IF R_HMICommand.Q THEN
    IF MainPMLControl_Simplified.ResetPressed AND
       MainPMLControl_Simplified.ResetPermissive AND
       MainPMLControl_Standard.CurrentState = E_PMLState.ePMLState_Aborted THEN
        ipModule.ChangeState(Tc3_PackML_V2.E_PMLCommand.ePMLCommand_Clear);
    ELSIF MainPMLControl_Simplified.ResetPressed AND MainPMLControl_Simplified.ResetPermissive THEN
        ipModule.ChangeState(Tc3_PackML_V2.E_PMLCommand.ePMLCommand_Reset);
    ELSIF MainPMLControl_Simplified.StartPressed AND MainPMLControl_Simplified.StartPermissive THEN
        IF MainPMLControl_Standard.CurrentState = Tc3_PackML_V2.E_PMLState.ePMLState_Idle THEN
            ipModule.ChangeState(Tc3_PackML_V2.E_PMLCommand.ePMLCommand_Start);
        ELSIF MainPMLControl_Standard.CurrentState = Tc3_PackML_V2.E_PMLState.ePMLState_Held THEN
            ipModule.ChangeState(Tc3_PackML_V2.E_PMLCommand.ePMLCommand_Unhold);
        ELSIF MainPMLControl_Standard.CurrentState = Tc3_PackML_V2.E_PMLState.ePMLState_Suspended THEN
            ipModule.ChangeState(Tc3_PackML_V2.E_PMLCommand.ePMLCommand_Unsuspend);
        END_IF
    ELSIF MainPMLControl_Simplified.StopPressed AND MainPMLControl_Simplified.StopPermissive THEN
        ipModule.ChangeState(Tc3_PackML_V2.E_PMLCommand.ePMLCommand_Stop);
    ELSIF MainPMLControl_Simplified.AbortPressed AND MainPMLControl_Simplified.AbortPermissive THEN
        ipModule.ChangeState(Tc3_PackML_V2.E_PMLCommand.ePMLCommand_Abort);
    ELSIF MainPMLControl_Simplified.HoldPressed AND MainPMLControl_Simplified.HoldPermissive THEN
        ipModule.ChangeState(Tc3_PackML_V2.E_PMLCommand.ePMLCommand_Hold);
    ELSIF ipModule.StateCommand <> MainPMLControl_Standard.StateCommand THEN
        ipModule.StateCommand := MainPMLControl_Standard.StateCommand;
    ELSIF ipModule.ModeCommand <> MainPMLControl_Standard.ModeCommand THEN
        ipModule.ModeCommand := MainPMLControl_Standard.ModeCommand;
    END_IF
END_IF

MainPMLControl_Simplified.StartPermissive := MainPMLControl_Standard.CurrentState = Tc3_PackML_V2.E_PMLState.ePMLState_Idle OR
                                             MainPMLControl_Standard.CurrentState = Tc3_PackML_V2.E_PMLState.ePMLState_Held OR
                                             MainPMLControl_Standard.CurrentState = Tc3_PackML_V2.E_PMLState.ePMLState_Suspended;

MainPMLControl_Simplified.HoldPermissive := MainPMLControl_Standard.CurrentState = Tc3_PackML_V2.E_PMLState.ePMLState_Execute OR
                                            MainPMLControl_Standard.CurrentState = Tc3_PackML_V2.E_PMLState.ePMLState_Unsuspending OR
                                            MainPMLControl_Standard.CurrentState = Tc3_PackML_V2.E_PMLState.ePMLState_Unholding;

MainPMLControl_Simplified.StopPermissive := MainPMLControl_Simplified.AbortPermissive :=
    MainPMLControl_Standard.CurrentState = Tc3_PackML_V2.E_PMLState.ePMLState_Held OR
    MainPMLControl_Standard.CurrentState = Tc3_PackML_V2.E_PMLState.ePMLState_Suspended OR
    MainPMLControl_Standard.CurrentState = Tc3_PackML_V2.E_PMLState.ePMLState_Idle;

MainPMLControl_Simplified.ResetPermissive := MainPMLControl_Standard.CurrentState = Tc3_PackML_V2.E_PMLState.ePMLState_Complete OR
                                             MainPMLControl_Standard.CurrentState = Tc3_PackML_V2.E_PMLState.ePMLState_Stopped OR
                                             MainPMLControl_Standard.CurrentState = Tc3_PackML_V2.E_PMLState.ePMLState_Aborted;
END_METHOD

PROPERTY Control : SPT_BaseTypes.I_PackML_Control
SET
ipModule := Control;
END_SET
END_PROPERTY

METHOD FINAL ModeChanged
VAR_INPUT
    NewMode : SPT_BaseTypes.E_PMLUnitMode;
END_VAR
MainPMLControl_Standard.ModeCommand := NewMode;
END_METHOD

METHOD FINAL StateChanged
VAR_INPUT
    NewState : SPT_BaseTypes.E_PMLCommand;
END_VAR
MainPMLControl_Standard.StateCommand := NewState;
END_METHOD

PROPERTY ForceHoldRequested : Bool
GET
ForceHoldRequested := (MainPMLControl_Standard.CurrentState = Tc3_PackML_V2.E_PMLState.ePMLState_Unsuspending OR
                      MainPMLControl_Standard.CurrentState = Tc3_PackML_V2.E_PMLState.ePMLState_Unholding) AND
                      MainPMLControl_Simplified.HoldPressed;
END_GET
END_PROPERTY

METHOD FINAL Initialize : BOOL
IF Registered THEN
    Initialize := TRUE;
END_IF
END_METHOD

PROPERTY Registered : BOOL
GET
Registered := ipModule <> 0;
END_GET
END_PROPERTY

END_FUNCTION_BLOCK

// Machine/EquipmentModules/Functional Layer/FB_Carriage
FUNCTION_BLOCK FB_Carriage EXTENDS FB_EquipmentModule_SR
VAR
    // Sub module definitions here

    // List of sub modules

    ipSubModules_Init : ARRAY[1..Parameters_PackML_Base.MAX_NO_OF_SUBMODULES] OF I_PackML_BaseModule := [];

    // Component definitions here

    // Transporter components based on class diagram

    Pos                 : FB_Component_BasicSlaveAxis_SoE := (Name := 'Position');
    Pick                : FB_Component_BasicSlaveAxis_SoE := (Name := 'Pick');
    BoardPresentSensor1 : FB_DigitalSensor                := (Name := 'BoardPresentSensor1');
    BoardPresentSensor2 : FB_DigitalSensor                := (Name := 'BoardPresentSensor2');
    HomingSensor        : FB_DigitalSensor                := (Name := 'HomingSensor');

    //Alarms for this module

    Pick_TorqueControl          : SPT_Motion_Control.MC_TorqueControl;
    Pick_HomingInfo             : ST_HomingParams;
    Pick_TorqueReference AT %Q* : UINT  := 100;
    Pick_First_Torque           : LREAL := -30;
    Pick_Second_Torque          : LREAL := -20;
    Pick_Home_Torque            : LREAL := 35;
    Pick_Lag                    : LREAL := 8;
    Pick_Vel                    : LREAL := 1200;

    MoveStates    : ST_MoveStates;
    SpeedSelected : E_SpeedOptions := E_SpeedOptions.TESTING1;

    Execute_TorqueMove      : BOOL;
    _SensorOverride         : BOOL;
    _SensorIgnore           : BOOL;
    BoardsIgnoredCount      : USINT;
    BoardSecured_AfterStop  : BOOL;
    GrabTorqueNotCompleting : BOOL;
    ReleaseNotFinished      : BOOL;
    MoveIdleNotFinished     : BOOL;
END_VAR

VAR CONSTANT
    //reports 

    FAULT : INT := 1;

    //Alarms

    UNWIND_ALARM_COUNT    : INT   := 5;
    CARRIAGE_ALARMS_COUNT : USINT := 10;
END_VAR

VAR
	PickMotorCmds_Extra : ST_MotorControls_NonStandard;
	PosMotorCmds_Extra : ST_MotorControls_NonStandard;

    _TargetPos       : LREAL;
    _IdlePos         : REAL;
    _HoldingBoard    : BOOL;
    _TestPick        : BOOL;
    _BoardSecured    : BOOL;
    _BoardDataToPass : ST_BoardData;

    _CarriageCollisionCheckOK    : BOOL;
    _BoardCollisionCheckOK       : BOOL;
    _MoveClearActive             : BOOL;
    _BoardHeight                 : LREAL;
    _MoveState                   : E_MoveCarriageState;
    _MoveSubState                : UDINT;
    CarriageMovementRequestState : UDINT;

    _ClearOfCarriages      : BOOL;
    _ClearOfBoards         : BOOL;
    _ActuatorsOpen         : BOOL;
    _ActuatorsClosed       : BOOL;
    _MovementRequested     : BOOL;
    _OpenActuatorsRequest  : BOOL;
    _CloseActuatorsRequest : BOOL;

    MoveIdleState : USINT;

    HomeHardStop : BOOL;

    //Homing Options

    TorqueOptions : SPT_Motion_Control.ST_TorqueControlOptions;

    _PressPermissions : ST_MediatorInterface;

    _MasterAxisRef : REFERENCE TO SPT_Motion_Control.AXIS_REF;
    _AxisRef       : REFERENCE TO SPT_Motion_Control.AXIS_REF;

    Grab_State    : E_GrabState;
    Release_State : E_ReleaseState;

    LastBoardHeightGrabbed : LREAL := 100;
    ;

    CarriageAlarms : ARRAY[1..CARRIAGE_ALARMS_COUNT] OF FB_TcAlarm;
	
END_VAR

METHOD CyclicLogic
VAR_INPUT
END_VAR
IF NOT _InitComplete THEN
    _InitComplete := Initialize();
    RETURN;
END_IF

SUPER^.CyclicLogic();

//HMI control for EM

fbControlSourceHMI.CyclicLogic();

//Set the current alarm severity for this module

// _CurrentAlarmSeverity := F_GetMaxSeverityRaised(Alarms:=UnwindAlarms, CurrentSeverity:=_CurrentAlarmSeverity);

IF _CurrentAlarmSeverity >= TcEventSeverity.Error THEN
    ChangeState(E_PMLCommand.ePMLCommand_Abort);
END_IF

IF _CurrentState <> E_PMLState.ePMLState_Unsuspending AND _CurrentState <> E_PMLState.ePMLState_Unholding THEN
    BoardSecured_AfterStop := FALSE;
END_IF

CyclicLogicSimulation();

BoardPresentSensor1.SimulationMode := E_SensorSimulationMode.InputDriven;
BoardPresentSensor2.SimulationMode := E_SensorSimulationMode.InputDriven;

BoardPresentSensor1.SimulationInput := TRUE;
BoardPresentSensor2.SimulationInput := TRUE;

Pos.Master1      REF= _MasterAxisRef;
Pos.RatioMaster1 := 1;

Pick_HomingInfo.HomePosMax := 284;
Pick_HomingInfo.HomePosMin := 84;

AllowHMIControl(ThisModuleOnly := FALSE);

IF testbool1 THEN
    IF TorqueHoming(Motor      := Pick,
                    HomingInfo := Pick_HomingInfo,
                    Velocity   := 100,
                    Torque     := 35,
                    Direction  := SPT_Motion_Control.MC_Direction.MC_Positive_Direction) THEN
        testbool1 := FALSE;
    END_IF
END_IF
END_METHOD

(*! @summary This method contains code which will execute when this PackML module is in the <b>Starting</b> state*)
METHOD PROTECTED Starting

VAR
    AllDone : bool;
END_VAR
CASE DescendantSequenceState OF
    0:
        IF MotorsInit() THEN
            DescendantSequenceState     := 10;
            MoveIdleState               := 0;
            Pick_HomingInfo.HomingState := 0;
        END_IF

    10:
        IF NOT _InSimulation THEN
            IF TorqueHoming(Motor      := Pick,
                            HomingInfo := Pick_HomingInfo,
                            Velocity   := 100,
                            Torque     := 35,
                            Direction  := SPT_Motion_Control.MC_Direction.MC_Positive_Direction) THEN
                DescendantSequenceState := 20;
            END_IF
        ELSE
            DescendantSequenceState := 20;
        END_IF

    20:
//         IF MoveIdleOnStarting() THEN
//             DescendantSequenceState := 30;
//         END_IF
// 
//     30:

        MoveStates.Grab    := 0;
        MoveStates.Release := 0;
        SUPER^.Starting();
END_CASE
END_METHOD

//! @summary This method contains code which will execute when this PackML module is in the <b>Unholding</b> state
METHOD PROTECTED Unholding
VAR
    i               : UDINT;
    SubModulesReady : BOOL := TRUE;
END_VAR

(*! <description><b></b><table> 
	<tr>
		<th> Previous State </th>
		<th> Transition In </th>
		<th> Transition Out </th>
		<th> Next State  </th> 
	</tr>
	<tr>
		<td> Held </td>
		<td> Unhold Command </td> 
		<td> State Complete </td>
		<td> Execute </td> 
	</tr>
</table>
This method is called as required by <c>StateControl()</c>
</description> 

*)
IF _ForceHold = FALSE THEN
    CASE _MotorInitState OF
        0:
            IF _ComponentsReset = FALSE THEN
                _ComponentsReset := ResetOnResume();
            ELSE
                _MotorInitState := 1;
            END_IF

        1:
            IF _MotorsHomed = FALSE THEN
                _MotorsHomed := MotorsHome();
            ELSE
                _MotorInitState := 2;
            END_IF

        2:
            IF _MotorsReset = FALSE THEN
                _MotorsReset := MotorsInit();
            ELSE
                _MotorInitState := 3;

            END_IF

        3:
            IF _AlignNeeded THEN
                IF MotorsInitAlignGearIn() THEN
                    _MotorInitState := 4;
                END_IF
            ELSE
                _MotorInitState := 4;
            END_IF

            Grab_State    := 0;
            Release_State := 0;

        4:
            IF _HoldingBoard THEN
                IF GrabBoard(LastBoardHeightGrabbed, SkipMoveAbs := TRUE) THEN
                    _MotorInitState := 5;
                END_IF

            ELSE
                IF ReleaseBoard() THEN
                    _MotorInitState := 5;
                END_IF
            END_IF

        5:
            FOR i := 1 TO NumberOfSubModules DO
                IF ipSubModules[i].CurrentState = E_PMLState.ePMLState_Held THEN
                    ipSubModules[i].StateCommand := ePMLCommand_Unhold;
                ELSIF ipSubModules[i].CurrentState = E_PMLState.ePMLState_Suspended THEN
                    ipSubModules[i].StateCommand := ePMLCommand_Unsuspend;
                END_IF
            END_FOR

            FOR i := 1 TO NumberOfSubModules DO
                SubModulesReady := SubModulesReady AND (ipSubModules[i].CurrentState = ePMLState_Execute);
            END_FOR

            IF SubModulesReady AND (StateTasksComplete OR NoStateTasksToComplete) THEN
                NoStateTasksToComplete := TRUE;
                StateTasksComplete     := FALSE;
                StateComplete();
            END_IF
    END_CASE
ELSE
    FOR i := 1 TO NumberOfSubModules DO
        IF ipSubModules[i].CurrentState = E_PMLState.ePMLState_Held THEN
            ipSubModules[i].StateCommand := ePMLCommand_Unhold;
        ELSIF ipSubModules[i].CurrentState = E_PMLState.ePMLState_Suspended THEN
            ipSubModules[i].StateCommand := ePMLCommand_Unsuspend;
        END_IF
    END_FOR

    FOR i := 1 TO NumberOfSubModules DO
        SubModulesReady := SubModulesReady AND (ipSubModules[i].CurrentState = ePMLState_Execute);
    END_FOR

    IF SubModulesReady AND (StateTasksComplete OR NoStateTasksToComplete) THEN
        NoStateTasksToComplete := TRUE;
        StateTasksComplete     := FALSE;
        StateComplete();
    END_IF
END_IF
END_METHOD

//! @summary This method contains code which will execute when this PackML module is in the <b>Unsuspending</b> state
METHOD PROTECTED Unsuspending
VAR
    i               : UDINT;
    SubModulesReady : BOOL := TRUE;
END_VAR

(*! <description><b></b><table> 
	<tr>
		<th> Previous State </th>
		<th> Transition In </th>
		<th> Transition Out </th>
		<th> Next State  </th> 
	</tr>
	<tr>
		<td> Suspended </td>
		<td> Unsuspend Command </td> 
		<td> State Complete </td>
		<td> Execute </td> 
	</tr>
</table>
This method is called as required by <c>StateControl()</c>
</description> 

*)
IF _ForceHold = FALSE THEN
    CASE _MotorInitState OF
        0:
            IF _ComponentsReset = FALSE THEN
                _ComponentsReset := ResetOnResume();
            ELSE
                _MotorInitState := 1;
            END_IF

        1:
            IF _MotorsHomed = FALSE THEN
                _MotorsHomed := MotorsHome();
            ELSE
                _MotorInitState := 2;
            END_IF

        2:
            IF _MotorsReset = FALSE THEN
                _MotorsReset := MotorsInit();
            ELSE
                _MotorInitState := 3;

            END_IF

        3:
            IF _AlignNeeded THEN
                IF MotorsInitAlignGearIn() THEN
                    _MotorInitState := 4;
                END_IF
            ELSE
                _MotorInitState := 4;
            END_IF

            Grab_State    := 0;
            Release_State := 0;

        4:
            IF _HoldingBoard THEN
                IF GrabBoard(LastBoardHeightGrabbed, SkipMoveAbs := TRUE) THEN
                    _MotorInitState := 5;
                END_IF

            ELSE
                IF ReleaseBoard() THEN
                    _MotorInitState := 5;
                END_IF
            END_IF

        5:
            FOR i := 1 TO NumberOfSubModules DO
                ipSubModules[i].StateCommand := ePMLCommand_Unsuspend;
            END_FOR

            FOR i := 1 TO NumberOfSubModules DO
                SubModulesReady := SubModulesReady AND (ipSubModules[i].CurrentState = ePMLState_Execute);
            END_FOR

            IF SubModulesReady AND (StateTasksComplete OR NoStateTasksToComplete) THEN
                NoStateTasksToComplete := TRUE;
                StateTasksComplete     := FALSE;
                StateComplete();
            END_IF
    END_CASE
ELSE
    FOR i := 1 TO NumberOfSubModules DO
        ipSubModules[i].StateCommand := ePMLCommand_Unsuspend;
    END_FOR

    FOR i := 1 TO NumberOfSubModules DO
        SubModulesReady := SubModulesReady AND (ipSubModules[i].CurrentState = ePMLState_Execute);
    END_FOR

    IF SubModulesReady AND (StateTasksComplete OR NoStateTasksToComplete) THEN
        NoStateTasksToComplete := TRUE;
        StateTasksComplete     := FALSE;
        StateComplete();
    END_IF
END_IF
END_METHOD

METHOD PROTECTED CreateEvents
VAR_INPUT
END_VAR
F_CreateAllEventsInClass(Alarms     := CarriageAlarms,
                         ClassSize  := SIZEOF(TC_EVENTS.Carriage),
                         pInitEvent := ADR(TC_EVENTS.Carriage.InitReferenceEvent),
                         Prefix     := _Name);

SUPER^.CreateEvents();
END_METHOD

METHOD GrabBoard : BOOL
VAR_INPUT
    BoardHeight : LREAL;
    SkipMoveAbs : BOOL := FALSE;
END_VAR

VAR
    result : USINT;
END_VAR

VAR_INST
    Previous_State : E_GrabState;
    AlarmTON       : TON;
END_VAR
GrabBoard := FALSE;

CASE Grab_State OF
    GRAB_START:
        MoveStates.Release := 0;
        _HoldingBoard      := TRUE;
        //Move to Initial Height

        Execute_TorqueMove := FALSE;
        _BoardSecured      := FALSE;

        IF SkipMoveAbs = FALSE OR _InSimulation THEN
            Pick.MoveAbsolute(BoardHeight + 25, TRUE);
            Grab_State := GRAB_MOVE_CHECK;
        ELSE
            Grab_State := GRAB_TORQUE;
        END_IF

        LastBoardHeightGrabbed := BoardHeight;
        AlarmTON(IN := FALSE, PT := T#5S);

    GRAB_MOVE_CHECK:
        IF Pick.InPosition AND NOT Pick.Busy THEN
            IF _TestPick OR _InSimulation THEN
                Grab_State := GRAB_FINISHED;
            ELSE
                Grab_State := GRAB_TORQUE;
            END_IF
        ELSIF Pick.Error THEN
            Grab_State := GRAB_ERROR;
        END_IF

    GRAB_TORQUE:
        TorqueOptions.EnableManualTorqueStartValue := TRUE;
        TorqueOptions.ManualTorqueStartValue       := Pick.Axis.NcToPlc.ActTorque;

        Pick_TorqueControl.Torque := Pick_First_Torque;
        Execute_TorqueMove        := TRUE;

        Trace('Pick Motor Torque Command High');

        IF ABS(Pick.Axis.NcToPlc.ActTorque - Pick_TorqueControl.Torque) < 0.5 AND Pick.Axis.NcToPlc.ActVelo < 0.2 THEN
            Grab_State         := GRAB_VERIFY;
            Execute_TorqueMove := FALSE;
        ELSIF Pick.Error THEN
            Grab_State := GRAB_ERROR;
        END_IF

        AlarmTON(IN := TRUE, PT := T#10S);
        GrabTorqueNotCompleting := AlarmTON.Q;

    GRAB_VERIFY:
        IF (BoardPresentSensor1.Active AND BoardPresentSensor2.Active) OR _SensorOverride OR _SensorIgnore OR SkipMoveAbs THEN
            Grab_State := GRAB_FINISHED;
        ELSE
            Grab_State := GRAB_ERROR;
        END_IF

    GRAB_ERROR:
		Pick.Disable();
        result := RaiseMessageBox(Header   := 'Wrong or missing board detected',
                                  Message1 := 'Carriage tried to stab board and one or both sensors are not being made',
                                  Message2 := 'Select Retry to try grabbing the board again',
                                  Message3 := 'Select Override to ignore sensor for this board',
                                  Message4 := 'Select Ignore to ignore sensors on pick for the next 10 boards',
                                  Btn1     := 'Retry',
                                  Btn3     := 'Override',
                                  Btn5     := 'Ignore');

        IF result = 1 THEN
            Grab_State := GRAB_RESUME_START;
        ELSIF result = 3 THEN
            _SensorOverride := TRUE;
            Grab_State      := GRAB_RESUME_START;
        ELSIF result = 5 THEN
            _SensorIgnore      := TRUE;
            BoardsIgnoredCount := 0;
            Grab_State         := GRAB_RESUME_START;
        END_IF

    GRAB_RESUME_START:
        IF _CurrentState = E_PMLState.ePMLState_Suspended THEN
            ChangeState(State := E_PMLCommand.ePMLCommand_Unsuspend);
        ELSIF _CurrentState = E_PMLState.ePMLState_Execute THEN
            Grab_State := GRAB_START;
        END_IF

    GRAB_FINISHED:

        _BoardSecured := TRUE;
        GrabBoard     := TRUE;
        Grab_State    := GRAB_START;
END_CASE

Pick_TorqueControl(Axis              := Pick.Axis,
                   Execute           := Execute_TorqueMove,
                   TorqueRamp        := 50,
                   VelocityLimitHigh := Pick_Vel,
                   VelocityLimitLow  := -Pick_Vel,
                   Options           := TorqueOptions);

IF Grab_State <> Previous_State THEN
    Trace(CONCAT('Carriage grab state change to: ', TO_STRING(Grab_State)));
END_IF

Previous_State := Grab_State;
END_METHOD

METHOD HMIControl
VAR_INPUT
END_VAR

VAR_INST
    HomeCommand_Pick     : BOOL;
    PowerOnCommand_Pick  : BOOL;
    PowerOffCommand_Pick : BOOL;
    PowerOnCommand_Pos   : BOOL;
    PowerOffCommand_Pos  : BOOL;
END_VAR
PickMotorCmds_Extra.Temp_R_Trig[1](CLK := PickMotorCmds_Extra.MotorCmd[1]);

PowerOnCommand_Pick := PickMotorCmds_Extra.Temp_R_Trig[1].Q AND PowerOnCommand_Pick = FALSE;

IF PowerOnCommand_Pick THEN
    IF Pick.Enable() THEN
        PowerOnCommand_Pick := FALSE;
    END_IF
END_IF

PickMotorCmds_Extra.Temp_R_Trig[2](CLK := PickMotorCmds_Extra.MotorCmd[2]);

PowerOffCommand_Pick := PickMotorCmds_Extra.Temp_R_Trig[2].Q AND PowerOffCommand_Pick = FALSE;

IF PowerOffCommand_Pick THEN
    IF Pick.Disable() THEN
        PowerOffCommand_Pick := FALSE;
    END_IF
END_IF

PickMotorCmds_Extra.Temp_R_Trig[3](CLK := PickMotorCmds_Extra.MotorCmd[3]);

HomeCommand_Pick := PickMotorCmds_Extra.Temp_R_Trig[3].Q AND HomeCommand_Pick = FALSE;

IF HomeCommand_Pick THEN
    IF TorqueHoming(Motor      := Pick,
                    HomingInfo := Pick_HomingInfo,
                    Velocity   := 100,
                    Torque     := 35,
                    Direction  := SPT_Motion_Control.MC_Direction.MC_Positive_Direction) THEN
        HomeCommand_Pick := FALSE;
    END_IF

END_IF



PosMotorCmds_Extra.Temp_R_Trig[1](CLK := PosMotorCmds_Extra.MotorCmd[1]);

PowerOnCommand_Pos := PosMotorCmds_Extra.Temp_R_Trig[1].Q AND PowerOnCommand_Pos = FALSE;

IF PowerOnCommand_Pos THEN
    IF Pos.Enable() THEN
        PowerOnCommand_Pos := FALSE;
    END_IF
END_IF

PosMotorCmds_Extra.Temp_R_Trig[2](CLK := PosMotorCmds_Extra.MotorCmd[2]);

PowerOnCommand_Pos := PosMotorCmds_Extra.Temp_R_Trig[2].Q AND PowerOnCommand_Pos = FALSE;

IF PowerOnCommand_Pos THEN
    IF Pos.Disable() THEN
        PowerOnCommand_Pos := FALSE;
    END_IF
END_IF
END_METHOD

//! @summary Basic module initialization logic
METHOD PROTECTED Initialize : BOOL;
VAR
    i                        : UDINT;
    varInfo                  : __SYSTEM.VAR_INFO;
    AllSubUnitsInitialized   : BOOL := TRUE;
    AllComponentsInitialized : BOOL := TRUE;
END_VAR

//! @description This method is called by <c>CyclicLogic()</c> as required
Initialize := FALSE;

CASE DescendantSequenceState OF
    0:
        RegisterComponent(Pos);
        RegisterComponent(Pick);
        RegisterComponent(BoardPresentSensor1);
        RegisterComponent(BoardPresentSensor2);
        RegisterComponent(HomingSensor);

        _LogModeChanges         := FALSE;
        _LogStateChanges        := FALSE;
        DescendantSequenceState := DescendantSequenceState + 10;

    10:
        //Setup Custom modes here

        (*CustomModes(eMode                          :=,
                    sName                          :=,
                    bDisableClearing               :=,
                    bDisableStarting               :=,
                    bDisableSuspended              :=,
                    bDisableStopping               :=,
                    bDisableAborting               :=,
                    bDisableHolding                :=,
                    bDisableHeld                   :=,
                    bDisableUnholding              :=,
                    bDisableSuspending             :=,
                    bDisableUnsuspending           :=,
                    bDisableResetting              :=,
                    bDisableIdle                   :=,
                    bDisableCompleting             :=,
                    bDisableComplete               :=,
                    bEnableUnitModeChangeStopped   :=,
                    bEnableUnitModeChangeIdle      :=,
                    bEnableUnitModeChangeSuspended :=,
                    bEnableUnitModeChangeExecute   :=,
                    bEnableUnitModeChangeAborted   :=,
                    bEnableUnitModeChangeHeld      :=,
                    bEnableUnitModeChangeComplete  :=,
                    bError                         =>,
                    nErrorId                       =>);*)

        DescendantSequenceState := DescendantSequenceState + 10;

    20:
        //Copy Mode names

        FOR i := 1 TO 3 DO
            ModeNames[i] := F_UnitModeToString(UDINT_TO_DINT(i));
        END_FOR

        RegisterExternalController(Controller := fbControlSourceHMI);
        fbControlSourceHMI.CyclicLogic();
        DescendantSequenceState := DescendantSequenceState + 10;

    30:
        //Call the Super

        IF SUPER^.Initialize() THEN
            DescendantSequenceState := DescendantSequenceState + 10;
        END_IF

    40:
        Initialize := TRUE;
END_CASE
END_METHOD

METHOD PROTECTED Monitoring
VAR_INPUT
END_VAR
///////////////////////////////////////////////////////////////////////////////
// 5.-12. Suspend warnings
///////////////////////////////////////////////////////////////////////////////
IF (NOT CarriageAlarms[E_Carriage.GrabTorqueNotFinished].bRaised) AND GrabTorqueNotCompleting THEN
    // Raise alarm if Infeed is taking a long time to get a board
    CarriageAlarms[E_Carriage.GrabTorqueNotFinished].Raise(0);
ELSIF CarriageAlarms[E_Carriage.GrabTorqueNotFinished].bRaised AND (NOT GrabTorqueNotCompleting) THEN
    // Clear when a board is found
    CarriageAlarms[E_Carriage.GrabTorqueNotFinished].Clear(0, 0);
END_IF;

IF (NOT CarriageAlarms[E_Carriage.GrabTorqueNotFinished].bRaised) AND ReleaseNotFinished THEN
    // Raise alarm if Infeed is taking a long time to get a board
    CarriageAlarms[E_Carriage.GrabTorqueNotFinished].Raise(0);
ELSIF CarriageAlarms[E_Carriage.GrabTorqueNotFinished].bRaised AND (NOT ReleaseNotFinished) THEN
    // Clear when a board is found
    CarriageAlarms[E_Carriage.GrabTorqueNotFinished].Clear(0, 0);
END_IF;

IF (NOT CarriageAlarms[E_Carriage.MoveIdleNotFinished].bRaised) AND MoveIdleNotFinished THEN
    // Raise alarm if Infeed is taking a long time to get a board
    CarriageAlarms[E_Carriage.MoveIdleNotFinished].Raise(0);
ELSIF CarriageAlarms[E_Carriage.MoveIdleNotFinished].bRaised AND (NOT MoveIdleNotFinished) THEN
    // Clear when a board is found
    CarriageAlarms[E_Carriage.MoveIdleNotFinished].Clear(0, 0);
END_IF;

//////////////////////////////////////////////////////////////////////////
// Wrap-up: Evaluate overall severity, then run the extended Monitoring
//////////////////////////////////////////////////////////////////////////
_CurrentAlarmSeverity := TcEventSeverity.Verbose;
_CurrentAlarmSeverity := F_GetMaxSeverityRaised(Alarms := CarriageAlarms, CurrentSeverity := _CurrentAlarmSeverity);

// Finally, run the extended monitoring
// SUPER^.Monitoring();
END_METHOD

METHOD MotorsInit : BOOL
VAR_INPUT
END_VAR
MotorsInit := FALSE;

IF _InSimulation THEN
    IF MotorResetAndEnable(Pos) AND MotorResetAndEnable(Pick) THEN
        MotorsInit := TRUE;
    END_IF
ELSE
    IF MotorResetAndEnable(Pos) AND MotorResetAndEnable(Pick) THEN
        MotorsInit := TRUE;
    END_IF
END_IF
END_METHOD

METHOD MoveIdleOnStarting : BOOL
VAR_INPUT
END_VAR

VAR_INST
    AlarmTON : TON;
END_VAR
MoveIdleOnStarting := FALSE;

CASE MoveIdleState OF
    0:
        _HoldingBoard := FALSE;
        //check to see if pick is retracted

        //TODO limit switch for carriage retract instead of position check

        IF ReleaseBoard() THEN
            MoveIdleState := 10;
        END_IF

        AlarmTON(IN := FALSE, PT := T#10S);

    10:
        // Move to Position

        Pos.MoveAbsolute(Position := _IdlePos, AbortPrevious := TRUE);
        MoveIdleState := 11;

    11:
        // verify position

        AlarmTON(IN := FALSE, PT := T#10S);

        IF Pos.Busy THEN
            MoveIdleState := 20;
        END_IF

        MoveIdleNotFinished := AlarmTON.Q;

    20:
        MoveStates.Idle    := 0;
        MoveIdleOnStarting := TRUE;

END_CASE
END_METHOD

METHOD ReleaseBoard : BOOL
VAR_INPUT
    Prep        : BOOL  := FALSE;
    PrepPickPos : LREAL := 0;
END_VAR

VAR_INST
    Previous_State : E_ReleaseState;
    AlarmTON       : TON;
    PreviousPos    : LREAL;
END_VAR
ReleaseBoard := FALSE;

CASE Release_State OF
    RELEASE_START:
        MoveStates.Grab := 0;
        _BoardSecured   := FALSE;
        //Move to Initial Height

        IF Pick.ActualPosition > 270 THEN
            Release_State := RELEASE_FINISHED;
        ELSE
            Release_State := RELEASE_MOVE;
        END_IF

        AlarmTON(IN := FALSE, PT := T#5S);

    RELEASE_MOVE:
        PreviousPos := Pick.ActualPosition;

        Pick.MoveAbsolute(275, TRUE);
        Release_State := RELEASE_MOVE_CHECK;

    RELEASE_MOVE_CHECK:
        AlarmTON(IN := TRUE, PT := T#5S);

        IF (Pick.InPosition AND NOT Pick.Busy) OR (Prep = TRUE AND Pick.Busy AND ABS(PreviousPos - Pick.ActualPosition) > 25) THEN
            Release_State   := RELEASE_FINISHED;
            _SensorOverride := FALSE;
            AlarmTON(IN := FALSE, PT := T#5S);

            IF _SensorIgnore = TRUE AND BoardsIgnoredCount > 10 THEN
                _SensorIgnore := FALSE;
            ELSE
                BoardsIgnoredCount := BoardsIgnoredCount + 1;
            END_IF
        END_IF

        ReleaseNotFinished := AlarmTON.Q;

    RELEASE_FINISHED:
        _HoldingBoard := FALSE;
        ReleaseBoard  := TRUE;
        Release_State := RELEASE_START;
END_CASE

IF Release_State <> Previous_State THEN
    Trace(CONCAT('Carriage release state change to: ', TO_STRING(Release_State)));
END_IF

Previous_State := Release_State;
END_METHOD

METHOD SetSpeeds : BOOL
VAR_INPUT
	PosVel : LREAL;
	PickVel : LREAL;
END_VAR
Pos.Velocity  := PosVel;
Pick.Velocity := PickVel;

Pick.Acceleration := Pick.Velocity * 8;
Pick.Deceleration := Pick.Velocity * 8;
Pos.Acceleration  := Pos.Velocity * 1.4;
Pos.Deceleration  := Pos.Velocity * 1.4;
END_METHOD

METHOD TestLengthPosCompare : BOOL
VAR_INPUT
END_VAR
TestLengthPosCompare := FALSE;
IF Pos.ActualPosition > (BEPoint_Backup.Infeed-38.1 + (60* 25.4)) THEN
    TestLengthPosCompare := TRUE;
END_IF
END_METHOD

METHOD ZPrepMove : BOOL
VAR_INPUT
	PrepPos : LREAL;
END_VAR
ZPrepMove := FALSE;
Pick.MoveAbsolute(PrepPos, TRUE);

IF Pick.Busy THEN
    ZPrepMove := TRUE;
END_IF
END_METHOD

PROPERTY ActuatorsClosed : bool
SET
_ActuatorsClosed := ActuatorsClosed;
END_SET
END_PROPERTY

PROPERTY ActuatorsOpen : bool
SET
_ActuatorsOpen := ActuatorsOpen;
END_SET
END_PROPERTY

PROPERTY AxisRef : REFERENCE TO SPT_Motion_Control.AXIS_REF;
GET
AxisRef REF= Pos.Axis;
END_GET
END_PROPERTY

PROPERTY BoardHeight : lreal
SET
_BoardHeight := BoardHeight;
END_SET
END_PROPERTY

PROPERTY BoardSecured : BOOL
GET
BoardSecured := _BoardSecured;
END_GET
SET
END_SET
END_PROPERTY

PROPERTY ClearOfBoards : bool
GET
ClearOfBoards := _ClearOfBoards;
END_GET
SET
_ClearOfBoards := ClearOfBoards;
END_SET
END_PROPERTY

PROPERTY ClearOfCarriages : bool
GET
ClearOfCarriages := _ClearOfCarriages;
END_GET
SET
_ClearOfCarriages := ClearOfCarriages;
END_SET
END_PROPERTY

PROPERTY CloseActuatorsRequest : bool
GET
CloseActuatorsRequest := _CloseActuatorsRequest;
END_GET
END_PROPERTY

PROPERTY HoldingBoard : Bool
GET
HoldingBoard := _HoldingBoard;
END_GET
END_PROPERTY

PROPERTY IdlePos : REAL
GET
IdlePos := _IdlePos;
END_GET
SET
_IdlePos := IdlePos;
END_SET
END_PROPERTY

PROPERTY IgnoreSensors : BOOL
GET
IgnoreSensors := _SensorIgnore;
END_GET
SET
_SensorIgnore := IgnoreSensors;
END_SET
END_PROPERTY

PROPERTY MasterAxis : REFERENCE TO SPT_Motion_Control.AXIS_REF;
SET
_MasterAxisRef REF= MasterAxis;
END_SET
END_PROPERTY

PROPERTY MoveClearActive : BOOL
GET
MoveClearActive := _MoveClearActive;
END_GET
SET
_MoveClearActive := MoveClearActive;
END_SET
END_PROPERTY

PROPERTY MovementRequested : bool
GET
MovementRequested := _MovementRequested;
END_GET
END_PROPERTY

PROPERTY MoveState : E_MoveCarriageState;
GET
MoveState := _MoveState;
END_GET
SET
_MoveState := MoveState;
END_SET
END_PROPERTY

PROPERTY MoveSubState : udint
GET
MoveSubState := _MoveSubState;
END_GET
SET
_MoveSubState := MoveSubState;
END_SET
END_PROPERTY

PROPERTY OpenActuatorsRequest : bool
GET
OpenActuatorsRequest := _OpenActuatorsRequest;
END_GET
END_PROPERTY

PROPERTY OverrideSensors : BOOL
GET
OverrideSensors := _SensorOverride;
END_GET
SET
_SensorOverride := OverrideSensors;
END_SET
END_PROPERTY

PROPERTY PressPermissions : REFERENCE TO ST_MediatorInterface
GET
PressPermissions REF= _PressPermissions;
END_GET
SET
_PressPermissions := PressPermissions;
END_SET
END_PROPERTY

PROPERTY Request_WS : E_WaitSync
SET
_RequestedWaitSync := Request_WS;
END_SET
END_PROPERTY

PROPERTY Response_WS : E_WaitSync
GET
Response_WS := _ResponseWaitSync;
END_GET
END_PROPERTY

PROPERTY TargetPos : LREAL
GET
TargetPos := _TargetPos;
END_GET
SET
_TargetPos := TargetPos;
END_SET
END_PROPERTY

END_FUNCTION_BLOCK

// Machine/EquipmentModules/Functional Layer/FB_Handoff
FUNCTION_BLOCK FB_Handoff EXTENDS FB_EquipmentModule_SR
VAR
    // Sub module definitions here

    // List of sub modules

    ipSubModules_Init : ARRAY[1..Parameters_PackML_Base.MAX_NO_OF_SUBMODULES] OF I_PackML_BaseModule := [];

    // Component definitions here

    CenteringClamp     : ARRAY[1..2] OF FB_DoubleSolenoidRetractFeedback := [(Name := 'Clamp_1'), (Name := 'Clamp_2')];
    BoardPresentSensor : FB_DigitalSensor                                := (Name := 'BoardPresentSensor');

    _ClampsClosed : BOOL;
END_VAR

VAR CONSTANT

    // Reports 

    FAULT : INT := 1;

    // Alarms

    PULL_WHEELS_ALARM_COUNT : INT := 5;
END_VAR

VAR
    _BoardDataToPass : ST_BoardData;
    _Location        : LREAL;
    _HoldingBoard    : BOOL;

    _ClampsOpen : BOOL;
END_VAR

METHOD CyclicLogic
VAR_INPUT
END_VAR
IF NOT _InitComplete THEN
    _InitComplete := Initialize();
    RETURN;
END_IF

SUPER^.CyclicLogic();

//HMI control for EM

fbControlSourceHMI.CyclicLogic();

//Set the current alarm severity for this module

// _CurrentAlarmSeverity := F_GetMaxSeverityRaised(Alarms:=PullWheelAlarms, CurrentSeverity:=_CurrentAlarmSeverity);

//Simulate Alarm Messaging

IF (CenteringClamp[1].InSimulation OR CenteringClamp[1].Retracted) AND (CenteringClamp[2].InSimulation OR CenteringClamp[2].Retracted) THEN
    _ClampsOpen := TRUE;
ELSE
    _ClampsOpen := FALSE;
END_IF

IF (CenteringClamp[1].InSimulation OR CenteringClamp[1].Extended) AND (CenteringClamp[2].InSimulation OR CenteringClamp[2].Extended) THEN
    _ClampsClosed := TRUE;
ELSE
    _ClampsClosed := FALSE;
END_IF

// CyclicLogicSimulation();
END_METHOD

METHOD GrabBoard : BOOL
VAR_INPUT
END_VAR
GrabBoard := FALSE;

FOR i := 1 TO 2 DO
    CenteringClamp[i].Extend();
END_FOR

IF CenteringClamp[1].Extended AND CenteringClamp[1].Extended THEN
    GrabBoard := TRUE;
    // 	Trace('Clamp Closed');
END_IF
END_METHOD

METHOD HMIControl
VAR_INPUT
END_VAR
IF HMI_INPUT[1] THEN
	FOR i := 1 TO 2 DO 
		ReleaseBoard(); 
	END_FOR
END_IF

IF HMI_INPUT[2] THEN
	FOR i := 1 TO 2 DO 
		GrabBoard(); 
	END_FOR
END_IF
END_METHOD

//! @summary Basic module initialization logic
METHOD PROTECTED Initialize : BOOL;
VAR
    i                        : UDINT;
    varInfo                  : __SYSTEM.VAR_INFO;
    AllSubUnitsInitialized   : BOOL := TRUE;
    AllComponentsInitialized : BOOL := TRUE;
END_VAR

//! @description This method is called by <c>CyclicLogic()</c> as required
Initialize := FALSE;

CASE DescendantSequenceState OF
    0:
        RegisterComponent(BoardPresentSensor);

        FOR i := 1 TO 2 DO
            RegisterComponent(CenteringClamp[i]);
        END_FOR

        _LogModeChanges         := FALSE;
        _LogStateChanges        := FALSE;
        DescendantSequenceState := DescendantSequenceState + 10;

    10:
        //Setup Custom modes here

        (*CustomModes(eMode                          :=,
                    sName                          :=,
                    bDisableClearing               :=,
                    bDisableStarting               :=,
                    bDisableSuspended              :=,
                    bDisableStopping               :=,
                    bDisableAborting               :=,
                    bDisableHolding                :=,
                    bDisableHeld                   :=,
                    bDisableUnholding              :=,
                    bDisableSuspending             :=,
                    bDisableUnsuspending           :=,
                    bDisableResetting              :=,
                    bDisableIdle                   :=,
                    bDisableCompleting             :=,
                    bDisableComplete               :=,
                    bEnableUnitModeChangeStopped   :=,
                    bEnableUnitModeChangeIdle      :=,
                    bEnableUnitModeChangeSuspended :=,
                    bEnableUnitModeChangeExecute   :=,
                    bEnableUnitModeChangeAborted   :=,
                    bEnableUnitModeChangeHeld      :=,
                    bEnableUnitModeChangeComplete  :=,
                    bError                         =>,
                    nErrorId                       =>);*)

        DescendantSequenceState := DescendantSequenceState + 10;

    20:
        //Copy Mode names

        FOR i := 1 TO 3 DO
            ModeNames[i] := F_UnitModeToString(UDINT_TO_DINT(i));
        END_FOR

        RegisterExternalController(Controller := fbControlSourceHMI);
        fbControlSourceHMI.CyclicLogic();
        DescendantSequenceState := DescendantSequenceState + 10;

    30:
        //Call the Super

        IF SUPER^.Initialize() THEN
            DescendantSequenceState := DescendantSequenceState + 10;
        END_IF

    40:
        Initialize := TRUE;
END_CASE
END_METHOD

METHOD ReleaseBoard : BOOL
VAR_INPUT
END_VAR
ReleaseBoard := FALSE;

FOR i := 1 TO 2 DO
    CenteringClamp[i].Retract();
END_FOR

IF CenteringClamp[1].Retracted AND CenteringClamp[1].Retracted THEN
    ReleaseBoard := TRUE;
    // 	Trace('Clamp Opened');
END_IF
END_METHOD

PROPERTY ClampsClosed : bool
GET
ClampsClosed := _ClampsClosed;
END_GET
END_PROPERTY

PROPERTY ClampsOpen : bool
GET
ClampsOpen := _ClampsOpen;
END_GET
END_PROPERTY

PROPERTY DisableClamp1 : BOOL
SET
CenteringClamp[1].InSimulation := DisableClamp1;
END_SET
END_PROPERTY

PROPERTY DisableClamp2 : BOOL
SET
CenteringClamp[2].InSimulation := DisableClamp2;
END_SET
END_PROPERTY

PROPERTY HoldingBoard : Bool
GET
HoldingBoard := _HoldingBoard;
END_GET
SET
_HoldingBoard := HoldingBoard;
END_SET
END_PROPERTY

PROPERTY Location : LREAL
GET
Location := _Location;
END_GET
SET
_Location := Location;
END_SET
END_PROPERTY

PROPERTY Request_WS : E_WaitSync
SET
_RequestedWaitSync := Request_WS;
END_SET
END_PROPERTY

PROPERTY Response_WS : E_WaitSync
GET
Response_WS := _ResponseWaitSync;
END_GET
END_PROPERTY

END_FUNCTION_BLOCK

// Machine/EquipmentModules/Functional Layer/FB_Infeed
FUNCTION_BLOCK FB_Infeed EXTENDS FB_EquipmentModule_SR
VAR
    // Sub module definitions here

    // List of sub modules

    ipSubModules_Init : ARRAY[1..Parameters_PackML_Base.MAX_NO_OF_SUBMODULES] OF I_PackML_BaseModule := [];

    // Component definitions here
    LengthCheckSensorMed  : FB_DigitalSensor := (Name := 'LengthCheckSensorLong');
    LengthCheckSensorLong  : FB_DigitalSensor := (Name := 'LengthCheckSensorLong');

    InfeedMotor        : FB_Component_ABB_VFD_EIP                                := (Name := 'InfeedMotor');
    Gate               : FB_DoubleSolenoidFeedback                       := (Name := 'Gate');
    CenteringClamp     : ARRAY[1..2] OF FB_DoubleSolenoidRetractFeedback := [(Name := 'Clamp_1'), (Name := 'Clamp_2')];
    BoardPresentSensor : FB_DigitalSensor                                := (Name := 'BoardPresentSensor');
    BoardEjectSensor   : FB_DigitalSensor                                := (Name := 'BoardEjectSensor');

    //Data for recipe

    _MoveClearActive                     : BOOL;
    _CarriageClearOfBoardPresentSensor   : BOOL;
    _IgnoreDoublePick                    : BOOL;
    _InfeedIgnoreDoublePick_Request      : BOOL;
    _InfeedIgnoreDoublePick_Acknowledged : BOOL;

    //Alarm Triggers

    InfeedTimeoutAlarm : BOOL;

    InfeedNotResettingAlarm : BOOL;
    _InfeedToInfeedRequest  : BOOL;
    _InfeedToInfeedReady    : BOOL;
    BoardRequested          : BOOL;
    BoardReleaseRequested   : BOOL;
    InfeedState_Simp        : E_INFEED_STATES;
END_VAR

VAR CONSTANT

    // Reports 

    FAULT : INT := 1;

    // Alarms

    PULL_WHEELS_ALARM_COUNT : INT   := 5;
    MinGearInLength         : REAL  := 3657.6;
    INFEED_ALARMS_COUNT     : USINT := 10;
END_VAR

VAR

    InfeedAlarms : ARRAY[1..INFEED_ALARMS_COUNT] OF FB_TcAlarm;

    InfeedState : E_Infeed_States;

    _CSVStep : REFERENCE TO ST_CSV_Step;

    _ReadyForBoard : BOOL;

    _CarriageTookBoard : BOOL;

    _StepComplete : BOOL;

    _BoardDropped : BOOL;

    _BoardCleardInfeed : BOOL;

    _BoardReadyForCarriage : BOOL;

    _TestExecute : BOOL;

    _clearinfeed : BOOL;

    Carriage1ReleaseRequest : BOOL;

    RequestBoard : BOOL;

    _BoardDataToPass : ST_BoardData;

    DataConfirmationNeeded : BOOL;

    DataConfirmationNeeded_State : USINT;

    _Carriage1ResetInfeed_Request : BOOL;

    _Carriage2ResetInfeed_Request : BOOL;

    DataReady : BOOL;

    _Debounce_Mode       : E_DebounceMode := E_DebounceMode.SimpleFlickerFilter;
    _Debounce_Time       : TIME           := T#1000MS;
    _Debounce_Time_Short : TIME           := T#500MS;

    _Sim_InfeedClear : BOOL;

    _LineNumber : INT;

	_ActiveInfeedMoving : BOOL;
	
    _CurrentParentState : E_PMLState;
	
	_Carriage1LengthTesting : BOOL;
END_VAR

METHOD CyclicLogic
VAR_INPUT
END_VAR

VAR
    testSensors : BOOL;
END_VAR
IF NOT _InitComplete THEN
    _InitComplete := Initialize();
    RETURN;
END_IF

//HMI control for EM
SUPER^.CyclicLogic();

fbControlSourceHMI.CyclicLogic();

//Set the current alarm severity for this module

// _CurrentAlarmSeverity := F_GetMaxSeverityRaised(Alarms:=PullWheelAlarms, CurrentSeverity:=_CurrentAlarmSeverity);

//Simulate Alarm Messaging

BoardEjectSensor.DebounceMode := _Debounce_Mode;
BoardEjectSensor.DebounceTime := _Debounce_Time;

BoardPresentSensor.DebounceMode := _Debounce_Mode;

IF THIS^.Name = 'Infeed_1' THEN
    BoardPresentSensor.DebounceTime := _Debounce_Time;

ELSIF THIS^.Name = 'Infeed_2' THEN
    BoardPresentSensor.DebounceTime := _Debounce_Time_Short;

END_IF

BoardPresentSensor.SimulationMode := E_SensorSimulationMode.InputDriven;
BoardEjectSensor.SimulationMode   := E_SensorSimulationMode.InputDriven;

IF InfeedState = INF_CONVEY AND _Sim_InfeedClear THEN
    BoardPresentSensor.SimulationInput := TRUE;
ELSIF InfeedState = INF_BOARD_PICKED_WS THEN
    BoardPresentSensor.SimulationInput := FALSE;
END_IF

IF _Carriage1LengthTesting THEN
    Gate.Retract();

    FOR i := 1 TO 2 DO
        CenteringClamp[i].Retract();
    END_FOR
END_IF

InfeedMotor.ReferenceVel := 2500;

Monitoring();
// CyclicLogicSimulation();
END_METHOD

(*! @summary This method contains code which will execute when this PackML module is in the <b>Holding</b> state*)
METHOD PROTECTED Aborting
InfeedMotor.Stop();
CenteringClamp[1].Retract();
CenteringClamp[2].Retract();
Gate.Retract();

SUPER^.Aborting();
END_METHOD

(*! @summary This method contains code which will execute when this PackML module is in the <b>Holding</b> state*)
METHOD PROTECTED Holding
InfeedMotor.Stop();

SUPER^.Holding();
END_METHOD

(*! @summary This method contains code which will execute when this PackML module is in the <b>Starting</b> state*)
METHOD PROTECTED Starting
DataConfirmationNeeded := TRUE;
_StepComplete          := FALSE;
DataReady              := FALSE;
_CarriageTookBoard     := FALSE;
_ReadyForBoard         := FALSE;
InfeedState            := INF_IDLE;

SUPER^.Starting();
END_METHOD

(*! @summary This method contains code which will execute when this PackML module is in the <b>Holding</b> state*)
METHOD PROTECTED Stopping
InfeedMotor.Stop();

SUPER^.Stopping();
END_METHOD

(*! @summary This method contains code which will execute when this PackML module is in the <b>Holding</b> state*)
METHOD PROTECTED Suspending
InfeedMotor.Stop();

SUPER^.Suspending();
END_METHOD

METHOD ExecuteStep : BOOL
VAR_INPUT
    Step : ST_CSV_Step;
END_VAR

VAR
    EmptyBoardData : ST_BoardData;
    tempDPLength   : LREAL;
END_VAR
ExecuteStep := FALSE;

CASE Step.seqName OF
    E_CommandName.Board:

        _BoardDataToPass.BoardID                 := Step.Details[1].Datas[1];
        _BoardDataToPass.BoardHeight             := STRING_TO_REAL(Step.Details[1].Datas[2]);
        _BoardDataToPass.BoardWidth              := STRING_TO_REAL(Step.Details[1].Datas[3]);
        _BoardDataToPass.BoardLength             := STRING_TO_REAL(Step.Details[1].Datas[4]);
        _BoardDataToPass.BoardNumber             := STRING_TO_INT(Step.Details[1].Datas[5]);
        _BoardDataToPass.LeadingEdgeBevelOffset  := STRING_TO_REAL(Step.Details[1].Datas[6]);
        _BoardDataToPass.TrailingEdgeBevelOffset := STRING_TO_REAL(Step.Details[1].Datas[7]);

        _BoardDataToPass.PickOffset :=
            MIN((_BoardDataToPass.LeadingEdgeBevelOffset +
                 ((_BoardDataToPass.BoardLength - _BoardDataToPass.LeadingEdgeBevelOffset - _BoardDataToPass.TrailingEdgeBevelOffset) / 2) -
                 (PICK_DEVICE_WIDTH / 2)),
                _BoardDataToPass.LeadingEdgeBevelOffset + DEFAULT_PICK_OFFSET);

        _BoardDataToPass.PickOffset := MIN(_BoardDataToPass.PickOffset, Global.BEPoint_Backup.Infeed - (Global.BEPoint_Backup.MinCarriagePos + 25));

        //TODO: calculate with leading/trailing offset eventually

        _BoardDataToPass.Positions[E_BoardData_Positions.CARRIAGE_1INFEED_HANDOFF].Position := Global.BEPoint_Backup.Infeed;
        _BoardDataToPass.Positions[E_BoardData_Positions.CARRIAGE_12_HANDOFF].Position      := BEPoint_Backup.PrePress + 100;

        _BoardDataToPass.DoublePickNeeded := _BoardDataToPass.BoardLength > Global.DOUBLEPICK_MIN_LENGTH;

        _BoardDataToPass.Positions[E_BoardData_Positions.GEAR_IN_SYNC].Position := (BEPoint_Backup.Infeed - 200) + _BoardDataToPass.BoardLength;

        IF _BoardDataToPass.BoardLength < 120 * 25.4 THEN
            _BoardDataToPass.Positions[E_BoardData_Positions.CARRIAGE_23_HANDOFF].Position := BEPoint_Backup.AssemblyHandoff + 100;
        ELSE
            _BoardDataToPass.Positions[E_BoardData_Positions.CARRIAGE_23_HANDOFF].Position := (BEPoint_Backup.PickPoint_1 - 630) + 100;
        END_IF

        _BoardDataToPass.Positions[E_BoardData_Positions.BOARD_DROP].Position := BEPoint_Backup.PickPoint_1 + (_BoardDataToPass.BoardLength / 2);

        DataReady := TRUE;

        IF _StepComplete THEN
            ExecuteStep        := TRUE;
            DataReady          := FALSE;
            _StepComplete      := FALSE;
            _CarriageTookBoard := FALSE;
        END_IF

ELSE
    DataReady        := FALSE;
    ExecuteStep      := TRUE;
    _BoardDataToPass := EmptyBoardData;
END_CASE
END_METHOD

METHOD PROTECTED Execute
VAR_INPUT
END_VAR

VAR
    WhiteLight : INT;
END_VAR
// Function based on mode.  NO need to make SUPER^.Executing() since it does nothing.
CASE _CurrentMode OF
    E_PMLUnitMode.ePMLUnitMode_Production:
        // Execute Logic
        IF THIS^.Name = 'Infeed_1' THEN
            Auto();
        ELSIF THIS^.Name = 'Infeed_2' THEN
            SuperSimpAuto();
        END_IF

    E_PMLUnitMode.ePMLUnitMode_Maintenance:
        ;

    E_PMLUnitMode.ePMLUnitMode_Manual:
        ;
END_CASE
END_METHOD

METHOD Auto : BOOL
VAR_INPUT
END_VAR

VAR
    result : USINT;
END_VAR

VAR_INST
    Previous_State           : E_Infeed_States;
    DoublePick_SubState      : E_Double_Pick_States;
    Previous_SubState        : E_Double_Pick_States;
    DoublePickSensorOverride : BOOL;
    IgnoreDP_F_TRIG          : F_TRIG;
    AlarmTON                 : TON;
END_VAR
// State Machine Logic
_ActiveInfeedMoving := FALSE;

IgnoreDP_F_TRIG(CLK := _InfeedIgnoreDoublePick_Request);

IF IgnoreDP_F_TRIG.Q THEN
    _InfeedIgnoreDoublePick_Acknowledged := FALSE;
END_IF

CASE InfeedState OF
    INF_IDLE: //IDLE
        AlarmTON(IN := TRUE, PT := T#5S);
        BoardRequested := FALSE;

        IF _CarriageTookBoard THEN
            _StepComplete := TRUE;
        ELSE
            IF NOT BoardEjectSensor.Active AND
               NOT BoardPresentSensor.Active AND
               _StepComplete = FALSE AND
               _MoveClearActive = FALSE AND
               DataReady = TRUE AND
               _BoardDataToPass.BoardID <> '' THEN
                InfeedState        := INF_CONVEY;
                _BoardCleardInfeed := TRUE;
                AlarmTON(IN := FALSE);
            END_IF
        END_IF

        InfeedNotResettingAlarm := AlarmTON.Q;

    INF_CONVEY: //Convey

        IF BoardRequested = FALSE AND _InSimulation = FALSE THEN
            AlarmTON(IN := FALSE);

            IF _LineNumber = 1 THEN
                //WS_MBI
                IF WaitSync_Handler(E_WaitSync.INFEED1_MBI_DROP_BOARD) THEN
                    BoardRequested := TRUE;
                END_IF
            ELSIF _LineNumber = 2 THEN
                //WS_Infeed2
                IF WaitSync_Handler(E_WaitSync.INFEED2_MBI_DROP_BOARD) THEN
                    BoardRequested := TRUE;
                END_IF
            END_IF
        ELSE
            AlarmTON(IN := TRUE, PT := T#20S);
            Gate.Extend();

            FOR i := 1 TO 2 DO
                CenteringClamp[i].Retract();
            END_FOR

            IF Gate.Extended AND CenteringClamp[1].Retracted AND CenteringClamp[2].Retracted THEN
                InfeedMotor.Jog(JogFW := TRUE);
                _ActiveInfeedMoving := TRUE;
            ELSE
                BoardPresentSensor.Reset();
            END_IF

            IF BoardPresentSensor.Active AND _CarriageClearOfBoardPresentSensor = TRUE THEN
                InfeedState := INF_BOARD_FOUND;
                AlarmTON(IN := FALSE);
            END_IF

            InfeedTimeoutAlarm := AlarmTON.Q;

            IF InfeedTimeoutAlarm THEN
                RaiseMessageBox(Header   := 'Board stuck in infeed',
                                Message1 := 'Board dropped in to infeed and is not moving forward',
                                Message2 := 'Manually push board forward to continue');
            END_IF
        END_IF

    INF_BOARD_FOUND: //Board Found
        FOR i := 1 TO 2 DO
            CenteringClamp[i].Extend();
        END_FOR

        IF InfeedMotor.Stop() AND CenteringClamp[1].Extended AND CenteringClamp[2].Extended THEN
            InfeedState := INF_BOARD_CHECK;
        END_IF

    INF_BOARD_CHECK: //Board Check?  
        IF BoardPresentSensor.Active THEN
            InfeedState := INF_ROUGH_LENGTH_CHECK;
        ELSE
            FOR i := 1 TO 2 DO
                CenteringClamp[i].Retract();
            END_FOR

            result := RaiseMessageBox(Header   := 'Board not found at Infeed!',
                                      Message1 := 'Infeed has secured a board and now it does not see a board',
                                      Message2 := 'Select Retry to start infeed again and pull board forward',
                                      Message3 := 'Select Override to tell carriage 1 to grab the board anyways',
                                      Message4 := 'WARNING if you get this message there is a potential sensor issue',
                                      Message5 := 'Check sensor at infeed to make sure its working properly',
                                      Message6 := 'If you select Retry from MBI it will drop a new board from MBI ',
                                      Btn1     := 'Retry',
                                      Btn2     := 'Retry from MBI',
                                      Btn3     := 'Override');

            IF result = 1 THEN
                InfeedState := INF_CONVEY;
            ELSIF result = 2 THEN
                BoardRequested := FALSE;
                InfeedState    := INF_CONVEY;
            ELSIF result = 3 THEN
                InfeedState := INF_ROUGH_LENGTH_CHECK;
            END_IF
        END_IF

    INF_ROUGH_LENGTH_CHECK: //Board Check?  
        IF RoughLengthCheck() OR _InSimulation THEN
            InfeedState := INF_BOARD_READY;
        ELSE
            FOR i := 1 TO 2 DO
                CenteringClamp[i].Retract();
            END_FOR

            result := RaiseMessageBox(Header   := 'Wrong board in Infeed conveyor',
                                      Message1 := CONCAT('Board expected: ', _BoardDataToPass.BoardID),
                                      Message2 := CONCAT('Length expected: ', LengthFormatString(_BoardDataToPass.BoardLength)),
                                      Message3 := 'Select Retry to start infeed again and pull board forward',
                                      Message4 := 'Select Override to tell carriage 1 to grab the board anyways',
                                      Message5 := 'WARNING if you get this message there is a potential sensor issue',
                                      Message6 := 'Check length sensors in the infeed to make sure its working properly',
                                      Message7 := 'If you select Retry from MBI it will drop a new board from MBI ',
                                      Btn1     := 'Retry',
                                      Btn2     := 'Retry from MBI',
                                      Btn3     := 'Override');

            IF result = 1 THEN
                InfeedState := INF_CONVEY;
            ELSIF result = 2 THEN
                BoardRequested := FALSE;
                InfeedState    := INF_CONVEY;
            ELSIF result = 3 THEN
                InfeedState := INF_BOARD_READY;
            END_IF
        END_IF

    INF_BOARD_READY: //Board Ready
        _InfeedToInfeedRequest := FALSE;
        _ReadyForBoard         := FALSE;

        FOR i := 1 TO 2 DO
            CenteringClamp[i].Extend();
        END_FOR

        IF CenteringClamp[1].Extended AND CenteringClamp[2].Extended THEN
            _BoardReadyForCarriage := TRUE;
            InfeedState            := INF_BOARD_READY_WS;
        END_IF

    INF_BOARD_READY_WS: // handshake with carriage 1 to let him know board's ready
        Gate.Retract();

        IF WaitSync_Handler(E_WaitSync.CARRIAGE1_INFEED_BOARD_READY) THEN
            InfeedState := INF_BOARD_PICKING_WS;
        END_IF

    INF_BOARD_PICKING_WS:
        Gate.Retract();

        IF WaitSync_Handler(E_WaitSync.CARRIAGE1_INFEED_PICKING) THEN
            InfeedState := INF_RETRACT_CLAMPS;
        END_IF

    INF_RETRACT_CLAMPS:
        Gate.Retract();

        FOR i := 1 TO 2 DO
            CenteringClamp[i].Retract();
        END_FOR

        IF CenteringClamp[1].Retracted AND CenteringClamp[2].Retracted AND Gate.Retracted THEN

            InfeedState := INF_BOARD_PICKED_WS;
        END_IF

    INF_BOARD_PICKED_WS: // last step on normal boards, DataConfirmationNeeded is the handshake for ExecuteStep to get new data
        IF WaitSync_Handler(E_WaitSync.CARRIAGE1_INFEED_BOARD_PICKED) THEN
            _CarriageTookBoard       := TRUE;
            _IgnoreDoublePick        := FALSE;
            DoublePickSensorOverride := FALSE;

            InfeedState := INF_BOARD_LENGTH_CHECK_CAR1;
        END_IF

    INF_BOARD_LENGTH_CHECK_CAR1:
        IF WaitSync_Handler(E_WaitSync.CARRIAGE1_INFEED_BOARD_LENGTH_CHECK) THEN
            IF _BoardDataToPass.DoublePickNeeded THEN
                InfeedState := INF_DOUBLE_PICK;
            ELSE
                InfeedState            := INF_IDLE;
                DataConfirmationNeeded := TRUE;
            END_IF
        ELSIF _Carriage1ResetInfeed_Request THEN
            InfeedState    := INF_CONVEY;
            BoardRequested := FALSE;
        END_IF

    INF_DOUBLE_PICK:
        // Carriage 1 needs to gear in and we don't want to bring any other boards forward

        IF NOT BoardEjectSensor.Active AND
           NOT BoardPresentSensor.Active AND
           DoublePickSensorOverride = FALSE AND
           _IgnoreDoublePick = FALSE AND
           _InSimulation = FALSE THEN
            //Board left when it shouldn't have, Wrong board loaded probably

            InfeedState := INF_WRONG_BOARD;
        ELSIF _InfeedIgnoreDoublePick_Request AND _InfeedIgnoreDoublePick_Acknowledged = FALSE THEN
            _InfeedIgnoreDoublePick_Acknowledged := TRUE;
            DoublePick_SubState                  := DP_REQUEST_WS;
            InfeedState                          := INF_IDLE;
            DataConfirmationNeeded               := TRUE;

        END_IF

        CASE DoublePick_SubState OF
            DP_REQUEST_WS:
                IF WaitSync_Handler(E_WaitSync.CARRIAGE2_INFEED_DOUBLE_PICK_REQUEST) THEN
                    IF _IgnoreDoublePick THEN
                        DoublePick_SubState    := DP_REQUEST_WS;
                        InfeedState            := INF_IDLE;
                        DataConfirmationNeeded := TRUE;
                    ELSE
                        DoublePick_SubState := DP_SECURE;
                    END_IF

                END_IF

            DP_SECURE:
                FOR i := 1 TO 2 DO
                    CenteringClamp[i].Extend();
                END_FOR

                IF CenteringClamp[1].Extended AND CenteringClamp[2].Extended THEN
                    DoublePick_SubState := DP_PICK_READY_WS;
                END_IF

            DP_PICK_READY_WS:
                IF WaitSync_Handler(E_WaitSync.CARRIAGE2_INFEED_DOUBLE_PICK_READY) THEN
                    DoublePick_SubState := DP_RETRACT_CLAMP;
                END_IF

            DP_RETRACT_CLAMP:
                FOR i := 1 TO 2 DO
                    CenteringClamp[i].Retract();
                END_FOR

                IF CenteringClamp[1].Retracted AND CenteringClamp[2].Retracted THEN
                    DoublePick_SubState := DP_PICK_DONE_WS;
                END_IF

            DP_PICK_DONE_WS:
                IF WaitSync_Handler(E_WaitSync.CARRIAGE2_INFEED_DOUBLE_PICK_DONE) THEN
                    DoublePick_SubState    := DP_REQUEST_WS;
                    InfeedState            := INF_IDLE;
                    DataConfirmationNeeded := TRUE;
                END_IF
        END_CASE

    INF_WRONG_BOARD:
        result := RaiseMessageBox(Header   := 'Wrong board detected',
                                  Message1 := 'Board should be long enough to still be in the infeed and needs double picked',
                                  Message2 := 'Select Retry to try check sensors again if board is still there',
                                  Message3 := 'Select Override to ignore sensors for this board and attempt double pick',
                                  Message4 := 'Select Ignore Double Pick to disable double pick for this board only',
                                  Message5 := 'WARNING overriding sensor or disable double pick could be missing nail plates',
                                  Message6 := 'WARNING if you override there is a potential for crashes',
                                  Btn1     := 'Retry',
                                  Btn3     := 'Override',
                                  Btn5     := 'Ignore Double Pick');

        IF result = 1 THEN
            InfeedState := INF_DOUBLE_PICK;
        ELSIF result = 3 THEN
            InfeedState              := INF_DOUBLE_PICK;
            DoublePickSensorOverride := TRUE;
        ELSIF result = 5 THEN
            InfeedState       := INF_DOUBLE_PICK;
            _IgnoreDoublePick := TRUE;
        END_IF

        //Wrong board error message needed here, reset to restart infeed

    999: //Error

END_CASE;

IF InfeedState <> Previous_State THEN
    Trace(CONCAT('Infeed state change to: ', TO_STRING(InfeedState)));
END_IF

Previous_State := InfeedState;

IF DoublePick_SubState <> Previous_SubState THEN
    Trace(CONCAT('Infeed double pick state change to: ', TO_STRING(DoublePick_SubState)));
END_IF

Previous_SubState := DoublePick_SubState;
END_METHOD

METHOD ClearInfeed : BOOL
VAR_INPUT
END_VAR
ClearInfeed := FALSE;
Gate.Retract();
InfeedMotor.Stop();

FOR i := 1 TO 2 DO
    CenteringClamp[i].Retract();
END_FOR

IF Gate.Retracted AND CenteringClamp[1].Retracted AND CenteringClamp[2].Retracted THEN
    ClearInfeed := TRUE;
END_IF
END_METHOD

METHOD PROTECTED CreateEvents
VAR_INPUT
END_VAR
F_CreateAllEventsInClass(Alarms     := InfeedAlarms,
                         ClassSize  := SIZEOF(TC_EVENTS.Infeed),
                         pInitEvent := ADR(TC_EVENTS.Infeed.InitReferenceEvent),
                         Prefix     := _Name);

SUPER^.CreateEvents();
END_METHOD

METHOD HMIControl
VAR_INPUT
END_VAR
IF HMI_INPUT[1] THEN
    Gate.Extend();
END_IF

IF HMI_INPUT[2] THEN
    Gate.Retract();
END_IF

IF HMI_INPUT[3] THEN
    FOR i := 1 TO 2 DO
        CenteringClamp[i].Extend();
    END_FOR
END_IF

IF HMI_INPUT[4] THEN
    FOR i := 1 TO 2 DO
        CenteringClamp[i].Retract();
    END_FOR
END_IF
END_METHOD

//! @summary Basic module initialization logic
METHOD PROTECTED Initialize : BOOL;
VAR
    i                        : UDINT;
    varInfo                  : __SYSTEM.VAR_INFO;
    AllSubUnitsInitialized   : BOOL := TRUE;
    AllComponentsInitialized : BOOL := TRUE;
END_VAR

//! @description This method is called by <c>CyclicLogic()</c> as required
Initialize := FALSE;

CASE DescendantSequenceState OF
    0:
        RegisterComponent(InfeedMotor);
        RegisterComponent(Gate);
        RegisterComponent(BoardPresentSensor);
        RegisterComponent(BoardEjectSensor);

        RegisterComponent(LengthCheckSensorMed);
        RegisterComponent(LengthCheckSensorLong);

        FOR i := 1 TO 2 DO
            RegisterComponent(CenteringClamp[i]);
        END_FOR

        _LogModeChanges         := FALSE;
        _LogStateChanges        := FALSE;
        DescendantSequenceState := DescendantSequenceState + 10;

    10:
        //Setup Custom modes here

        (*CustomModes(eMode                          :=,
                    sName                          :=,
                    bDisableClearing               :=,
                    bDisableStarting               :=,
                    bDisableSuspended              :=,
                    bDisableStopping               :=,
                    bDisableAborting               :=,
                    bDisableHolding                :=,
                    bDisableHeld                   :=,
                    bDisableUnholding              :=,
                    bDisableSuspending             :=,
                    bDisableUnsuspending           :=,
                    bDisableResetting              :=,
                    bDisableIdle                   :=,
                    bDisableCompleting             :=,
                    bDisableComplete               :=,
                    bEnableUnitModeChangeStopped   :=,
                    bEnableUnitModeChangeIdle      :=,
                    bEnableUnitModeChangeSuspended :=,
                    bEnableUnitModeChangeExecute   :=,
                    bEnableUnitModeChangeAborted   :=,
                    bEnableUnitModeChangeHeld      :=,
                    bEnableUnitModeChangeComplete  :=,
                    bError                         =>,
                    nErrorId                       =>);*)

        DescendantSequenceState := DescendantSequenceState + 10;

    20:
        //Copy Mode names

        FOR i := 1 TO 3 DO
            ModeNames[i] := F_UnitModeToString(UDINT_TO_DINT(i));
        END_FOR

        RegisterExternalController(Controller := fbControlSourceHMI);
        fbControlSourceHMI.CyclicLogic();
        DescendantSequenceState := DescendantSequenceState + 10;

    30:
        //Call the Super

        IF SUPER^.Initialize() THEN
            DescendantSequenceState := DescendantSequenceState + 10;
        END_IF

    40:
        Initialize := TRUE;
END_CASE
END_METHOD

METHOD PROTECTED Monitoring
VAR_INPUT
END_VAR
///////////////////////////////////////////////////////////////////////////////
// 5. Timeout: ID=5
///////////////////////////////////////////////////////////////////////////////
IF (NOT InfeedAlarms[E_Infeed.InfeedTimeout].bRaised) AND InfeedTimeoutAlarm THEN
    // Raise alarm if Infeed is taking a long time to get a board
    InfeedAlarms[E_Infeed.InfeedTimeout].Raise(0);
ELSIF InfeedAlarms[E_Infeed.InfeedTimeout].bRaised AND (NOT InfeedTimeoutAlarm) THEN
    // Clear when a board is found
    InfeedAlarms[E_Infeed.InfeedTimeout].Clear(0, 0);
END_IF;

///////////////////////////////////////////////////////////////////////////////
// 6. Timeout: ID=6
///////////////////////////////////////////////////////////////////////////////
IF (NOT InfeedAlarms[E_Infeed.InfeedNotResetting].bRaised) AND InfeedNotResettingAlarm THEN
    // Raise alarm if Infeed is taking too long to reset and start conveying
    InfeedAlarms[E_Infeed.InfeedNotResetting].Raise(0);
ELSIF InfeedAlarms[E_Infeed.InfeedNotResetting].bRaised AND (NOT InfeedNotResettingAlarm) THEN
    // Clear when infeed can convey forward
    InfeedAlarms[E_Infeed.InfeedNotResetting].Clear(0, 0);
END_IF;

//////////////////////////////////////////////////////////////////////////
// Wrap-up: Evaluate overall severity, then run the extended Monitoring
//////////////////////////////////////////////////////////////////////////
_CurrentAlarmSeverity := TcEventSeverity.Verbose;
_CurrentAlarmSeverity := F_GetMaxSeverityRaised(Alarms := InfeedAlarms, CurrentSeverity := _CurrentAlarmSeverity);

// Finally, run the extended monitoring
// SUPER^.Monitoring();
END_METHOD

METHOD ParseBoardData : BOOL
END_METHOD

METHOD RoughLengthCheck : BOOL
VAR_INPUT
END_VAR
RoughLengthCheck := FALSE;

IF _BoardDataToPass.BoardLength > BOARD_LENGTH_SENSOR2_LOCATION THEN
    IF LengthCheckSensorLong.Active AND LengthCheckSensorMed.Active THEN
        RoughLengthCheck := TRUE;
    ELSE
        RoughLengthCheck := FALSE;
    END_IF
ELSIF _BoardDataToPass.BoardLength > BOARD_LENGTH_SENSOR1_LOCATION THEN
    IF NOT LengthCheckSensorLong.Active AND LengthCheckSensorMed.Active THEN
        RoughLengthCheck := TRUE;
    ELSE
        RoughLengthCheck := FALSE;
    END_IF
ELSE
    IF NOT LengthCheckSensorLong.Active AND NOT LengthCheckSensorMed.Active THEN
        RoughLengthCheck := TRUE;
    ELSE
        RoughLengthCheck := FALSE;
    END_IF
END_IF
END_METHOD

METHOD SimpAuto : BOOL
VAR_INPUT
END_VAR

VAR
    result : USINT;
END_VAR

VAR_INST
    Previous_State           : E_Infeed_States;
    DoublePickSensorOverride : BOOL;
    InfeedToInfeedTrig       : R_TRIG;
    InfeedToInfeedConfirmed  : BOOL;
    AlarmTON                 : TON;

    BoardPresentTimeOff_TON : TON;
END_VAR
// State Machine Logic

CASE InfeedState_Simp OF
    INF_IDLE: //IDLE
        AlarmTON(IN := TRUE, PT := T#5S);
        BoardPresentTimeOff_TON(IN := NOT BoardPresentSensor.Active, PT := T#5S);
        _InfeedToInfeedReady := FALSE;
        BoardRequested       := FALSE;

        IF BoardPresentTimeOff_TON.Q THEN
            InfeedState_Simp := INF_CONVEY;
            _ReadyForBoard   := TRUE;
            AlarmTON(IN := FALSE);
        END_IF

        InfeedNotResettingAlarm := AlarmTON.Q;

    INF_CONVEY: //Convey

        IF BoardRequested = FALSE THEN
            IF WaitSync_Handler(E_WaitSync.INFEED2_MBI_DROP_BOARD) THEN
                BoardRequested := TRUE;
            END_IF
        ELSE
            BoardPresentTimeOff_TON(IN := FALSE, PT := T#5S);
            AlarmTON(IN := TRUE, PT := T#10S);

            _ReadyForBoard := TRUE;

            Gate.Extend();

            IF Gate.Extended THEN
                InfeedMotor.Jog(JogFW := TRUE);
            END_IF

            IF BoardPresentSensor.Active THEN
                InfeedState_Simp := INF_BOARD_FOUND;
                AlarmTON(IN := FALSE);
            END_IF

            InfeedTimeoutAlarm := AlarmTON.Q;

        END_IF

    INF_BOARD_FOUND: //Board Found

        IF InfeedMotor.Stop() THEN
            InfeedState_Simp := INF_BOARD_CHECK;
        END_IF

    INF_BOARD_CHECK:
        _ReadyForBoard := FALSE;
        Gate.Retract();

        IF Gate.Retracted AND BoardPresentSensor.Active THEN
            InfeedState_Simp := INF_BOARD_READY;
        END_IF

    INF_BOARD_READY: //Board Ready
        _ReadyForBoard := FALSE;
        Gate.Retract();
        _InfeedToInfeedReady := TRUE;

        IF BoardReleaseRequested = FALSE THEN
            IF THIS^.Name = 'Infeed_2' THEN
                IF WaitSync_Handler(E_WaitSync.INFEED1_INFEED2_RELEASE_BOARD) THEN
                    BoardReleaseRequested := TRUE;
                END_IF
            END_IF
        END_IF

        IF BoardReleaseRequested THEN

            InfeedMotor.Jog(JogFW := TRUE);

            IF BoardPresentSensor.Active = FALSE THEN
                InfeedState_Simp      := INF_IDLE;
                BoardReleaseRequested := FALSE;
            END_IF
        END_IF

    999: //Error

END_CASE;

IF InfeedState_Simp <> Previous_State THEN
    Trace(CONCAT('Infeed state change to: ', TO_STRING(InfeedState_Simp)));
END_IF

Previous_State := InfeedState_Simp;
END_METHOD

METHOD SuperSimpAuto : BOOL
VAR_INPUT
END_VAR
// State Machine Logic

CASE InfeedState_Simp OF
    INF_IDLE: //IDLE
		InfeedMotor.Stop();
        IF _ActiveInfeedMoving THEN
            InfeedState_Simp := INF_CONVEY;
        END_IF
		
    INF_CONVEY: //Convey

        Gate.Retract();

        IF Gate.Retracted then
            InfeedMotor.Jog(JogFW := TRUE);
        END_IF
		
		IF NOT _ActiveInfeedMoving THEN
            InfeedState_Simp := INF_IDLE;
		END_IF
END_CASE;
END_METHOD

PROPERTY ActiveInfeedMoving : Bool
GET
ActiveInfeedMoving := _ActiveInfeedmoving;
END_GET
SET
_ActiveInfeedMoving := ActiveInfeedmoving;
END_SET
END_PROPERTY

PROPERTY BoardDataToPass : ST_BoardData
GET
BoardDataToPass := _BoardDataToPass;
END_GET
END_PROPERTY

PROPERTY BoardDropped : bool
SET
_BoardDropped := BoardDropped;
END_SET
END_PROPERTY

PROPERTY BoardReadyForCarriage : bool
GET
BoardReadyForCarriage := _BoardReadyForCarriage;
END_GET
END_PROPERTY

PROPERTY Carriage1LengthTesting : bool
SET
_Carriage1LengthTesting := Carriage1LengthTesting;
END_SET
END_PROPERTY

PROPERTY Carriage1ResetInfeed_Request : bool
SET
_Carriage1ResetInfeed_Request := Carriage1ResetInfeed_Request;
END_SET
END_PROPERTY

PROPERTY Carriage2_DoublePickCancel_Request : bool
SET
_InfeedIgnoreDoublePick_Request := Carriage2_DoublePickCancel_Request;
END_SET
END_PROPERTY

PROPERTY Carriage2ResetInfeed_Request : bool
SET
_Carriage2ResetInfeed_Request := Carriage2ResetInfeed_Request;
END_SET
END_PROPERTY

PROPERTY CarriageClearOfBoardPresentSensor : bool
SET
_CarriageClearOfBoardPresentSensor := CarriageClearOfBoardPresentSensor;
END_SET
END_PROPERTY

PROPERTY IgnoreDoublePick : BOOL
GET
IgnoreDoublePick := _IgnoreDoublePick;
END_GET
END_PROPERTY

PROPERTY InfeedToInfeedReady : Bool
GET
InfeedToInfeedReady := _InfeedToInfeedReady;
END_GET
SET
_InfeedToInfeedReady := InfeedToInfeedReady;
END_SET
END_PROPERTY

PROPERTY InfeedToInfeedRequest : Bool
GET
InfeedToInfeedRequest := _InfeedToInfeedRequest;
END_GET
SET
_InfeedToInfeedRequest := InfeedToInfeedRequest;
END_SET
END_PROPERTY

PROPERTY LineNumber : INT
SET
_LineNumber := LineNumber;
END_SET
END_PROPERTY

PROPERTY MoveClearActive : BOOL
SET
_MoveClearActive := MoveClearActive;
END_SET
END_PROPERTY

PROPERTY ParentState : E_PMLState
SET
_CurrentParentState := ParentState;
END_SET
END_PROPERTY

PROPERTY ReadyForBoard : BOOL
GET
ReadyForBoard := _ReadyForBoard;
END_GET
END_PROPERTY

PROPERTY Sim_InfeedClear : bool
SET
_Sim_InfeedClear := Sim_InfeedClear;
END_SET
END_PROPERTY

PROPERTY TestExecute : bool
SET
_TestExecute := TestExecute;
END_SET
END_PROPERTY

END_FUNCTION_BLOCK

// Machine/EquipmentModules/Functional Layer/FB_MBI
FUNCTION_BLOCK FB_MBI EXTENDS FB_EquipmentModule_SR
VAR
    // Sub module definitions here

    // List of sub modules

    ipSubModules_Init : ARRAY[1..Parameters_PackML_Base.MAX_NO_OF_SUBMODULES] OF I_PackML_BaseModule := [];

    // Component definitions here

    InfeedMotor         : FB_Component_ABB_VFD_EIP            := (Name := 'InfeedMotor');
    IndexSensor         : FB_DigitalSensor            := (Name := 'IndexSensor');
    BoardPresentSensor1 : FB_DigitalSensor            := (Name := 'BoardPresentSensor1');
    BoardPresentSensor2 : FB_DigitalSensor            := (Name := 'BoardPresentSensor2');
    ControlPendant      : FB_ControlPendant           := (Name := 'ControlPendent');
    LightStack          : FB_Component_StackLight_MBI := (Name := 'LightStack');

    testErrorFlag       : BOOL;
    testErrorID         : UDINT;
    MBIInfeedHSTimeout  : BOOL;
    _MainSafetyOK       : BOOL;
    _CurrentParentState : E_PMLState;
    BoardDropRequested  : BOOL;
END_VAR

VAR
    _ActiveConvState : E_MBI_States;

    _BoardDropped     : BOOL := FALSE; // Flag indicating if a board was dropped   
    _DropBoard        : BOOL := FALSE; // Command to drop a board
    _bMonitorRearEdge : BOOL := FALSE; // Flag to monitor carriage rear edge

    // State machine variables

    _Active            : BOOL := FALSE;
    _ReadyForBoard     : BOOL; // The current input signal for ready for board.
    _ReadyForBoardPrev : BOOL := FALSE; // Holds the previous state of ReadyForBoard.
    _RisingEdgeReady   : BOOL := FALSE; // Indicates a rising edge detection.
    _bFoundBoardToDrop : BOOL; // The current input signal for ready for board.
    _bBoardInNextLane  : BOOL;
    _SubStep           : INT;
    _ResetActive       : BOOL;

    _TestExecute : BOOL;

    ReadyForBoard_RTRIG : R_TRIG;
    MBIAlarms           : ARRAY[1..MBI_ALARMS_COUNT] OF FB_TcAlarm;

    _LineNumber : INT;

END_VAR

VAR CONSTANT
    MBI_ALARMS_COUNT : USINT := 10;
END_VAR

VAR CONSTANT

    // Reports 

    FAULT : INT := 1;

    // Alarms

    PULL_WHEELS_ALARM_COUNT : INT := 5;

END_VAR

METHOD CyclicLogic
VAR_INPUT
END_VAR
IF NOT _InitComplete THEN
    _InitComplete := Initialize();
    RETURN;
END_IF

SUPER^.CyclicLogic();

//HMI control for EM
IF THIS^.Name = 'MBI_1' AND _LineNumber = 1 THEN
	LightStack.AmberLight.TurnOn();
	
ELSIF THIS^.Name = 'MBI_2' AND _LineNumber = 2 THEN
	LightStack.AmberLight.TurnOn();

ELSE
	LightStack.AmberLight.TurnOff();
END_IF
fbControlSourceHMI.CyclicLogic();

//Set the current alarm severity for this module

// _CurrentAlarmSeverity := F_GetMaxSeverityRaised(Alarms:=PullWheelAlarms, CurrentSeverity:=_CurrentAlarmSeverity);

//Simulate Alarm Messaging

CyclicLogicSimulation();

// Production();

Monitoring();

// ControlPendant.GreenButton.LED.Flash();

// ControlPendant.YellowButton.LED.Flash(T#300MS,T#500MS);

// ControlPendant.BlueButton.LED.Flash(T#700MS,T#500MS);
END_METHOD

(*! @summary This method contains code which will execute when this PackML module is in the <b>Holding</b> state*)
METHOD PROTECTED Aborting
InfeedMotor.Stop();

SUPER^.Aborting();
END_METHOD

(*! @summary This method contains code which will execute when this PackML module is in the <b>Holding</b> state*)
METHOD PROTECTED Holding
InfeedMotor.Stop();

SUPER^.Holding();
END_METHOD

(*! @summary This method contains code which will execute when this PackML module is in the <b>Starting</b> state*)
METHOD PROTECTED Starting
_ActiveConvState := 0;
_BoardDropped    := FALSE;

SUPER^.Starting();
END_METHOD

(*! @summary This method contains code which will execute when this PackML module is in the <b>Stopping</b> state*)
METHOD PROTECTED Stopping
InfeedMotor.Stop();

SUPER^.Stopping();
END_METHOD

(*! @summary This method contains code which will execute when this PackML module is in the <b>Holding</b> state*)
METHOD PROTECTED Suspending
InfeedMotor.Stop();

SUPER^.Suspending();
END_METHOD

(*! @summary This method contains code which will execute when this PackML module is in the <b>Unholding</b> state*)
METHOD PROTECTED Unholding
IF _MainSafetyOK THEN
    SUPER^.Unholding();
ELSE
    StateComplete();
END_IF
END_METHOD

(*! @summary This method contains code which will execute when this PackML module is in the <b>Unsuspending</b> state*)
METHOD PROTECTED Unsuspending
IF _MainSafetyOK THEN
    SUPER^.Unsuspending();
ELSE
    StateComplete();
END_IF
END_METHOD

(*! @summary This method contains code which will execute when this PackML module is in the <b>Aborted</b> state*)
METHOD PROTECTED Aborted
IF _MainSafetyOK THEN
    ChangeState(E_PMLCommand.ePMLCommand_Clear);
END_IF
END_METHOD

METHOD PROTECTED Execute
VAR_INPUT
END_VAR

VAR
    WhiteLight : INT;
END_VAR
// Function based on mode.  NO need to make SUPER^.Executing() since it does nothing.
IF _MainSafetyOK THEN
    IF ControlPendant.YellowButton.Button_Pressed THEN
        ChangeState(E_PMLCommand.ePMLCommand_Hold);
    END_IF

    IF ControlPendant.Mode_Auto THEN
        // Auto Mode Operations
        IF _CurrentParentState = E_PMLState.ePMLState_Execute THEN
            Auto();
            LightStack.WhiteLight.TurnOn();
        ELSE
            LightStack.WhiteLight.Flash();
            InfeedMotor.Stop();
        END_IF
    ELSIF ControlPendant.Mode_Manual_1 THEN
        // Manual Mode Forward Operations
        IF _MainSafetyOK THEN
            LightStack.WhiteLight.Flash();
            ManualMode_Forward();
        END_IF
    ELSIF ControlPendant.Mode_Manual_2 THEN
        // Manual Mode Reverse Operations

        IF _MainSafetyOK THEN
            LightStack.WhiteLight.Flash();
            ManualMode_Reverse();
        END_IF
    ELSE
        // Error Handling for No Mode Chosen

        InfeedMotor.Stop();
    END_IF
ELSE
    ChangeState(E_PMLCommand.ePMLCommand_Suspend);
END_IF

IF ControlPendant.Mode_Manual_1 OR ControlPendant.Mode_Manual_2 THEN
    ControlPendant.GreenButton.LED.TurnOff();
    ControlPendant.BlueButton.LED.TurnOn();
    ControlPendant.YellowButton.LED.TurnOn();
    _ActiveConvState := 0;
ELSIF ControlPendant.Mode_Auto THEN
    ControlPendant.GreenButton.LED.TurnOff();
    ControlPendant.BlueButton.LED.TurnOff();
    ControlPendant.YellowButton.LED.TurnOn();
ELSE
    ControlPendant.GreenButton.LED.TurnOn();
    ControlPendant.BlueButton.LED.TurnOn();
    ControlPendant.YellowButton.LED.TurnOn();
END_IF
END_METHOD

METHOD PROTECTED Held
VAR_INPUT
END_VAR
_ActiveConvState := acIDLE;

IF _MainSafetyOK THEN
    IF ControlPendant.GreenButton.Button_Pressed THEN
        ChangeState(E_PMLCommand.ePMLCommand_Unhold);
    END_IF

    ControlPendant.GreenButton.LED.TurnOn();
    ControlPendant.BlueButton.LED.TurnOff();
    ControlPendant.YellowButton.LED.TurnOff();
ELSE
    ControlPendant.GreenButton.LED.Flash();
    ControlPendant.BlueButton.LED.Flash();
    ControlPendant.YellowButton.LED.Flash();
END_IF
END_METHOD

METHOD PROTECTED Idle
VAR_INPUT
END_VAR
_ActiveConvState := acIDLE;

IF _MainSafetyOK THEN
    IF ControlPendant.GreenButton.Button_Pressed THEN
        ChangeState(E_PMLCommand.ePMLCommand_Start);
    END_IF

    ControlPendant.GreenButton.LED.TurnOn();
    ControlPendant.BlueButton.LED.TurnOff();
    ControlPendant.YellowButton.LED.TurnOff();
ELSE
    ControlPendant.GreenButton.LED.Flash();
    ControlPendant.BlueButton.LED.Flash();
    ControlPendant.YellowButton.LED.Flash();
END_IF
END_METHOD

METHOD PROTECTED Stopped
VAR_INPUT
END_VAR
IF _MainSafetyOK THEN
    ChangeState(E_PMLCommand.ePMLCommand_Reset);
END_IF
END_METHOD

METHOD PROTECTED Suspended
VAR_INPUT
END_VAR
_ActiveConvState := acIDLE;

IF _MainSafetyOK THEN
    IF ControlPendant.GreenButton.Button_Pressed THEN
        ChangeState(E_PMLCommand.ePMLCommand_Unsuspend);
    END_IF

    ControlPendant.GreenButton.LED.TurnOn();
    ControlPendant.BlueButton.LED.TurnOff();
    ControlPendant.YellowButton.LED.TurnOff();
ELSE
    ControlPendant.GreenButton.LED.Flash();
    ControlPendant.BlueButton.LED.Flash();
    ControlPendant.YellowButton.LED.Flash();
END_IF
END_METHOD

METHOD Auto : BOOL
VAR_INPUT
END_VAR

VAR_INST
    Previous_State : E_MBI_States;
    BoardDropTON   : TON;
END_VAR

VAR
    result : USINT;
END_VAR
// State Machine Logic

IF _ResetActive THEN
    _ActiveConvState := acIDLE;
ELSE
    CASE _ActiveConvState OF

        acIDLE:

            // Reset state machine variables

            _SubStep := 0;

            IF BoardPresentSensor2.Active THEN
                _bBoardInNextLane := FALSE;
                _ActiveConvState  := acWAIT_INFEED_READY;
            ELSE
                _ActiveConvState := acINDEX_FORWARD;
            END_IF

            BoardDropTON(IN := FALSE, PT := T#30S);

        acINDEX_FORWARD:

            // Index the conveyor forward until the first board sensor is made

            InfeedMotor.Jog(JogFW := TRUE);
            InfeedMotor.ReferenceVel := 2000;

            IF BoardPresentSensor2.Active THEN
                _ActiveConvState := acWAIT_INFEED_READY;
            END_IF

        acWAIT_INFEED_READY:
            // Board is in position, wait for infeed to be ready

            BoardDropTON(IN := TRUE, PT := T#30S);
            InfeedMotor.Stop();

            IF BoardDropRequested = FALSE THEN
                IF THIS^.Name = 'MBI_1' THEN
                    IF WaitSync_Handler(E_WaitSync.INFEED1_MBI_DROP_BOARD) THEN
                        BoardDropRequested := TRUE;
                    END_IF
                ELSIF THIS^.Name = 'MBI_2' THEN
                    IF WaitSync_Handler(E_WaitSync.INFEED2_MBI_DROP_BOARD) THEN
                        BoardDropRequested := TRUE;
                    END_IF
                END_IF
            END_IF

            IF BoardDropRequested THEN
                _ActiveConvState := acDUMP_BOARD;
                BoardDropTON(IN := FALSE, PT := T#30S);
            ELSE
                MBIInfeedHSTimeout := BoardDropTON.Q;
            END_IF

        acDUMP_BOARD:

            BoardDropRequested := FALSE;
            // Move forward to dump board

            InfeedMotor.Jog(JogFW := TRUE);

            CASE _SubStep OF
                0:
                    IF BoardPresentSensor2.Active THEN
                        _SubStep := 1;
                    END_IF

                1:
                    IF NOT BoardPresentSensor2.Active THEN
                        _ActiveConvState  := acIDLE;
                        _SubStep          := 0;
                        _BoardDropped     := TRUE;
                        _bMonitorRearEdge := FALSE;
                    END_IF

            END_CASE

        acBOARD_LOST:

        // TODO: Add error handling for board lost scenario
    END_CASE

END_IF

IF _ActiveConvState <> Previous_State THEN
    Trace(CONCAT('MBI state change to: ', TO_STRING(_ActiveConvState)));
END_IF

Previous_State := _ActiveConvState;
END_METHOD

METHOD PROTECTED CreateEvents
VAR_INPUT
END_VAR
F_CreateAllEventsInClass(Alarms     := MBIAlarms,
                         ClassSize  := SIZEOF(TC_EVENTS.MBI),
                         pInitEvent := ADR(TC_EVENTS.MBI.InitReferenceEvent),
                         Prefix     := _Name);

SUPER^.CreateEvents();
END_METHOD

METHOD HMIControl
VAR_INPUT
END_VAR
END_METHOD

//! @summary Basic module initialization logic
METHOD PROTECTED Initialize : BOOL;
VAR
    i                        : UDINT;
    varInfo                  : __SYSTEM.VAR_INFO;
    AllSubUnitsInitialized   : BOOL := TRUE;
    AllComponentsInitialized : BOOL := TRUE;
END_VAR

//! @description This method is called by <c>CyclicLogic()</c> as required
Initialize := FALSE;

CASE DescendantSequenceState OF
    0:
        RegisterComponent(InfeedMotor);
        RegisterComponent(BoardPresentSensor1);
        RegisterComponent(BoardPresentSensor2);
        RegisterComponent(IndexSensor);
        RegisterComponent(ControlPendant);
        RegisterComponent(LightStack);

        _LogModeChanges         := FALSE;
        _LogStateChanges        := FALSE;
        DescendantSequenceState := DescendantSequenceState + 10;

    10:
        //Setup Custom modes here

        (*CustomModes(eMode                          :=,
                    sName                          :=,
                    bDisableClearing               :=,
                    bDisableStarting               :=,
                    bDisableSuspended              :=,
                    bDisableStopping               :=,
                    bDisableAborting               :=,
                    bDisableHolding                :=,
                    bDisableHeld                   :=,
                    bDisableUnholding              :=,
                    bDisableSuspending             :=,
                    bDisableUnsuspending           :=,
                    bDisableResetting              :=,
                    bDisableIdle                   :=,
                    bDisableCompleting             :=,
                    bDisableComplete               :=,
                    bEnableUnitModeChangeStopped   :=,
                    bEnableUnitModeChangeIdle      :=,
                    bEnableUnitModeChangeSuspended :=,
                    bEnableUnitModeChangeExecute   :=,
                    bEnableUnitModeChangeAborted   :=,
                    bEnableUnitModeChangeHeld      :=,
                    bEnableUnitModeChangeComplete  :=,
                    bError                         =>,
                    nErrorId                       =>);*)

        DescendantSequenceState := DescendantSequenceState + 10;

    20:
        //Copy Mode names

        FOR i := 1 TO 3 DO
            ModeNames[i] := F_UnitModeToString(UDINT_TO_DINT(i));
        END_FOR

        RegisterExternalController(Controller := fbControlSourceHMI);
        fbControlSourceHMI.CyclicLogic();
        DescendantSequenceState := DescendantSequenceState + 10;

    30:
        //Call the Super

        IF SUPER^.Initialize() THEN
            DescendantSequenceState := DescendantSequenceState + 10;
        END_IF

    40:
        Initialize := TRUE;
END_CASE
END_METHOD

METHOD ManualMode_Forward : BOOL
VAR_INPUT
END_VAR
// State Machine Logic

InfeedMotor.ReferenceVel := 2000;

IF _ResetActive THEN
    _ActiveConvState := acIDLE;

ELSE
    IF ControlPendant.BlueButton.Button_Pressed AND NOT BoardPresentSensor2.Active THEN
        InfeedMotor.Jog(JogFW := TRUE);
    ELSE
        InfeedMotor.Stop();
    END_IF

END_IF
END_METHOD

METHOD ManualMode_Reverse : BOOL
VAR_INPUT
END_VAR
// State Machine Logic

InfeedMotor.ReferenceVel := -2000;

IF _ResetActive THEN
    _ActiveConvState := acIDLE;

ELSE
    IF ControlPendant.BlueButton.Button_Pressed THEN
        InfeedMotor.Jog(JogFW := TRUE);
    ELSE
        InfeedMotor.Stop();
    END_IF

END_IF
END_METHOD

METHOD PROTECTED Monitoring
VAR_INPUT
END_VAR
///////////////////////////////////////////////////////////////////////////////
// 5. Timeout: ID=5
///////////////////////////////////////////////////////////////////////////////
IF (NOT MBIAlarms[E_MBI.BoardNotDropping].bRaised) AND MBIInfeedHSTimeout THEN
    // Raise alarm if Infeed is taking a long time to get a board
    MBIAlarms[E_MBI.BoardNotDropping].Raise(0);
ELSIF MBIAlarms[E_MBI.BoardNotDropping].bRaised AND (NOT MBIInfeedHSTimeout) THEN
    // Clear when a board is found
    MBIAlarms[E_MBI.BoardNotDropping].Clear(0, 0);
END_IF;

//////////////////////////////////////////////////////////////////////////
// Wrap-up: Evaluate overall severity, then run the extended Monitoring
//////////////////////////////////////////////////////////////////////////
_CurrentAlarmSeverity := TcEventSeverity.Verbose;
_CurrentAlarmSeverity := F_GetMaxSeverityRaised(Alarms := MBIAlarms, CurrentSeverity := _CurrentAlarmSeverity);

// Finally, run the extended monitoring
// SUPER^.Monitoring();
END_METHOD

METHOD Production : BOOL
VAR_INPUT
END_VAR
ReadyForBoard_RTRIG(CLK := _ReadyForBoard);

IF ReadyForBoard_RTRIG.Q THEN
    _BoardDropped := FALSE;
END_IF

IF _ResetActive THEN
    InfeedMotor.Stop();
    _ActiveConvState := acIDLE;

    IF ControlPendant.GreenButton.Button_Pressed THEN
        _ResetActive := FALSE;
    END_IF
ELSE
    IF ControlPendant.Mode_Auto THEN
        // Auto Mode Operations
        IF _CurrentState = E_PMLState.ePMLState_Execute AND _MainSafetyOK THEN
            Auto();
        ELSE
            InfeedMotor.Stop();
        END_IF
    ELSIF ControlPendant.Mode_Manual_1 THEN
        // Manual Mode Forward Operations
        IF _MainSafetyOK THEN
            LightStack.WhiteLight.Flash();
            ManualMode_Forward();
        END_IF
    ELSIF ControlPendant.Mode_Manual_2 THEN
        // Manual Mode Reverse Operations

        IF _MainSafetyOK THEN
            LightStack.WhiteLight.Flash();
            ManualMode_Reverse();
        END_IF
    ELSE
        // Error Handling for No Mode Chosen

        InfeedMotor.Stop();
    END_IF

END_IF

// Light Stack Indicators

IF NOT ControlPendant.KeySwitch_Auto.Active OR (_ActiveConvState <> acWAIT_READY AND _ActiveConvState <> acDUMP_BOARD) THEN
    LightStack.WhiteLight.Flash();
    LightStack.AmberLight.TurnOff();
ELSE
    LightStack.WhiteLight.TurnOff();
    LightStack.AmberLight.TurnOn();
END_IF

IF _ResetActive THEN
    ControlPendant.GreenButton.LED.TurnOn();
    ControlPendant.BlueButton.LED.TurnOff();
    ControlPendant.YellowButton.LED.TurnOff();

ELSIF ControlPendant.Mode_Manual_1 OR ControlPendant.Mode_Manual_2 THEN
    ControlPendant.GreenButton.LED.TurnOff();
    ControlPendant.BlueButton.LED.TurnOn();
    ControlPendant.YellowButton.LED.TurnOn();
    _ActiveConvState := 0;
ELSIF ControlPendant.Mode_Auto THEN
    ControlPendant.GreenButton.LED.TurnOff();
    ControlPendant.BlueButton.LED.TurnOff();
    ControlPendant.YellowButton.LED.TurnOn();
ELSE
    ControlPendant.GreenButton.LED.Flash();
    ControlPendant.BlueButton.LED.Flash();
    ControlPendant.YellowButton.LED.Flash();

END_IF
END_METHOD

PROPERTY BoardDropped : bool
GET
BoardDropped := _BoardDropped;
END_GET
END_PROPERTY

PROPERTY LineNumber : INT
SET
_LineNumber := LineNumber;
END_SET
END_PROPERTY

PROPERTY MainSafetyOK : bool
SET
_MainSafetyOK := MainSafetyOK;
END_SET
END_PROPERTY

PROPERTY ParentState : E_PMLState
SET
_CurrentParentState := ParentState;
END_SET
END_PROPERTY

PROPERTY ReadyForBoard : BOOL
SET
_ReadyForBoard := ReadyForBoard;
END_SET
END_PROPERTY

PROPERTY TestExecute : bool
SET
_TestExecute := TestExecute;
END_SET
END_PROPERTY

END_FUNCTION_BLOCK

// Machine/EquipmentModules/Functional Layer/FB_Outfeed_Jig
FUNCTION_BLOCK FB_Outfeed_Jig EXTENDS FB_EquipmentModule_SR
VAR
    // Sub module definitions here

    // List of sub modules

    ipSubModules_Init : ARRAY[1..Parameters_PackML_Base.MAX_NO_OF_SUBMODULES] OF I_PackML_BaseModule := [];

    // Component definitions here

    Convey_Motors : ARRAY[1..7] OF FB_Conveyor;

    //Convey_Sensors        : ARRAY[1..7] OF FB_DigitalSensor;
    Shift_Motors   : FB_Component_ABB_VFD_EC;
    ControlPendant : FB_ControlPendant_Outfeed   := (Name := 'ControlPendent');
    LightStack     : FB_Component_StackLight_MBI := (Name := 'LightStack');

    //Alarms for this module

    AllDone                  : BOOL;
    testnum                  : INT   := 1;
    testpos                  : LREAL := 1000;
    testdist                 : LREAL := 1000;
    _PickPlace_Ready_ENUM    : E_WaitSync;
    _PickPlace_Done_ENUM     : E_WaitSync;
    MoveVelocitySpeed        : LREAL := -500;
    ClearOccupiedOutfeedData : BOOL;

    _OutfeedAutostopOK   : BOOL;
    SuspendTON           : TON;
    RecoveryDetected     : BOOL;
    IndexingBlockedAlarm : BOOL;
    TestConveyorsON      : BOOL;
    _ParentState         : E_PMLState;

    AllStopped                  : BOOL;
    EnableManualConveyorControl : BOOL;
    ManualConveyorSpeed         : LREAL := 500;
    ManualModeActive            : BOOL;
    ManualControlConveyFWD      : BOOL;
    ManualControlConveyREV      : BOOL;

    ManualReset : BOOL;
END_VAR

VAR CONSTANT
    OUTFEED_ALARMS_COUNT : USINT := 10;
END_VAR

VAR
    OutfeedJigAlarms : ARRAY[1..OUTFEED_ALARMS_COUNT] OF FB_TcAlarm;

    SimHomingLocalState : DINT;
    SimHomingIndex      : UDINT;

    OutfeedMasterAutoSpeed   : LREAL := 500;
    OutfeedMasterManualSpeed : LREAL := 50;

    TrussInfo         : ST_TrussInfo;
    IndexConveyor     : ST_IndexConveyor;
    PickPlace         : ST_PickPlace;
    _MaxConveyorCount : UDINT;
    _MainSafetyOK     : BOOL;
    _AutostopOK       : BOOL;

    //
    StartUp : BOOL := TRUE;

    _OutfeedConveyorStatus : ST_OutfeedConveyorStatus;
END_VAR

VAR PERSISTENT
    ConvData : ARRAY[1..7] OF ST_ConveyorData;
END_VAR

METHOD CyclicLogic
VAR_INPUT
END_VAR

VAR

END_VAR
IF NOT _InitComplete THEN
    _InitComplete := Initialize();
    RETURN;
END_IF

SUPER^.CyclicLogic();

FOR i := 1 TO _MaxConveyorCount DO
    ConvData[i].ConveyorID        := CONCAT('Conveyor No: ', UDINT_TO_STRING(i));
    ConvData[i].ConveyorStateStr  := TO_STRING(ConvData[i].State);
    ConvData[i].ActualPosition    := Convey_Motors[i].ActualPosition;
    ConvData[i].CurrentTruss      := ConvData[i].TrussInfo.TrussID;
    Convey_Motors[i].Velocity     := OutfeedMasterAutoSpeed;
    Convey_Motors[i].Acceleration := OutfeedMasterAutoSpeed * 2;
    Convey_Motors[i].Deceleration := OutfeedMasterAutoSpeed * 2;

END_FOR

_OutfeedConveyorStatus.Total    := _MaxConveyorCount;
_OutfeedConveyorStatus.Occupied := 0;

FOR i := _MaxConveyorCount TO 1 BY -1 DO
    IF ConvData[i].State = E_Outfeed_Conveyor_State.OCCUPIED OR
       ConvData[i].State = E_Outfeed_Conveyor_State.RECEIVING OR
       (i = 1 AND ConvData[i].State = E_Outfeed_Conveyor_State.BUILD_IN_PROGRESS) OR
       (i = 1 AND ConvData[i].State = E_Outfeed_Conveyor_State.INDEX_PREP) OR
       (i = _MaxConveyorCount AND ConvData[i].State = E_Outfeed_Conveyor_State.RESET) OR
       (i = _MaxConveyorCount AND ConvData[i].State = E_Outfeed_Conveyor_State.AUTO_RETRACT) THEN
        _OutfeedConveyorStatus.Occupied := _OutfeedConveyorStatus.Occupied + 1;
    END_IF
END_FOR

IF _CurrentState <> E_PMLState.ePMLState_Suspended THEN
    SuspendTON(IN := FALSE, PT := T#2S);

END_IF

IF ClearOccupiedOutfeedData THEN
    FOR i := 1 TO _MaxConveyorCount DO

        IF i = _MaxConveyorCount THEN
            ConvData[i].State := E_Outfeed_Conveyor_State.IDLE;
        ELSE
            ConvData[i].State := E_Outfeed_Conveyor_State.RESET;

        END_IF

        ClearOccupiedOutfeedData := FALSE;
    END_FOR
END_IF

Monitoring();
END_METHOD

(*! @summary This method contains code which will execute when this PackML module is in the <b>Suspending</b> state*)
METHOD PROTECTED Suspending
FOR i := 1 TO _MaxConveyorCount DO
    Convey_Motors[i].Stop();
END_FOR

SUPER^.Suspending();
END_METHOD

(*! @summary This method contains code which will execute when this PackML module is in the <b>Unsuspending</b> state*)
METHOD PROTECTED Unsuspending
IF _OutfeedAutostopOK AND _MainSafetyOK THEN
    SUPER^.Unsuspending();
ELSE
    StateComplete();
END_IF
END_METHOD

METHOD ExecuteStep : BOOL
VAR_INPUT
    Step : ST_CSV_Step;
END_VAR

VAR CONSTANT
    PICK_DEVICE_WIDTH   : LREAL := 203;
    DEFAULT_PICK_OFFSET : LREAL := 200;
END_VAR
ExecuteStep := FALSE;

CASE Step.seqName OF
    E_CommandName.TrussInfo:
        TrussInfoParse(Step, TrussInfo);
        ExecuteStep := RunTrussInfo();

    E_CommandName.PickPlace:
        PickPlaceParse(Step, PickPlace);
        ExecuteStep := RunPickPlace(PickPlace);

    E_CommandName.IndexConveyor:
        IndexConveyorParse(Step, IndexConveyor);
        ExecuteStep := RunIndexConveyor();

    E_CommandName.AssemblyEnd:
        ExecuteStep := IndexFull();

ELSE
    ExecuteStep := TRUE;

END_CASE
END_METHOD

METHOD RunIndexConveyor : BOOL
VAR_INPUT
END_VAR

VAR_INST
    SubState : UDINT;
END_VAR
IF Convey_Motors[1].Enabled AND Convey_Motors[1].Error = FALSE THEN
    IF IndexConveyor.ConvIndex MOD 2 = 0 THEN
        RunIndexConveyor := IndexHalf();

    ELSIF IndexConveyor.ConvIndex MOD 2 = 1 THEN
        RunIndexConveyor := IndexFull();

    END_IF
ELSE
    MotorResetAndEnable(Convey_Motors[1]);
END_IF
END_METHOD

METHOD RunPickPlace : BOOL
VAR_INPUT
    BoardData : reference to ST_PickPlace;
END_VAR

VAR
    result : USINT;
END_VAR

VAR_INST
    State : UDINT;
END_VAR
CASE State OF
    0:
        IF RecoveryDetected OR (BoardData.Number = 1 AND ConvData[1].State = E_Outfeed_Conveyor_State.BUILD_IN_PROGRESS) THEN
            result := RaiseMessageBox(Header   := 'Old truss data detected',
                                      Message1 := 'Conveyor has data from previous truss',
                                      Message2 := 'Select Clear if conveyor is clear and ready for current truss',
                                      Message3 := 'Select Index to send old truss out down the line',
                                      Message4 := 'WARNING make sure conveyor is clear or has correct truss on it',
                                      Message5 := 'If Index is pressed robot will place once truss is clear',
                                      Btn1     := 'Clear',
                                      Btn3     := 'Index');

            IF result = 1 THEN
                ConvData[1].State := E_Outfeed_Conveyor_State.IDLE;
                RecoveryDetected  := FALSE;
            ELSIF result = 3 THEN
                ConvData[1].State := E_Outfeed_Conveyor_State.INDEX_PREP;
                RecoveryDetected  := FALSE;
            END_IF
        ELSE
            IF BoardData.Number = 1 THEN
                IF ConvData[1].State = E_Outfeed_Conveyor_State.IDLE THEN
                    IF WaitSync_Handler(_PickPlace_Ready_ENUM) THEN
                        ConvData[1].State := E_Outfeed_Conveyor_State.BUILD_IN_PROGRESS;
                        State             := 1;
                    END_IF
                END_IF
            ELSE
                IF ConvData[1].State = E_Outfeed_Conveyor_State.BUILD_IN_PROGRESS OR ConvData[1].State = E_Outfeed_Conveyor_State.IDLE THEN
                    IF WaitSync_Handler(_PickPlace_Ready_ENUM) THEN
                        State             := 1;
                        ConvData[1].State := E_Outfeed_Conveyor_State.BUILD_IN_PROGRESS;
                    END_IF
                END_IF
            END_IF
        END_IF

    1:
        IF ConvData[1].State = E_Outfeed_Conveyor_State.BUILD_IN_PROGRESS THEN
            IF WaitSync_Handler(_PickPlace_Done_ENUM) THEN
                State := 2;
            END_IF
        END_IF

    2:
        FOR i := 1 TO 50 DO
            IF ConvData[1].BoardsPresent[i].ID = '' AND ConvData[1].BoardsPresent[i].Length = 0 THEN
                ConvData[1].BoardsPresent[i] := BoardData;
                EXIT;
            END_IF
        END_FOR

        ConvData[1].TrussInfo := TrussInfo;
        RunPickPlace          := TRUE;
        State                 := 0;

END_CASE
END_METHOD

METHOD RunTrussInfo : BOOL
VAR_INPUT
END_VAR

VAR
    i              : USINT;
    EmptyBoardData : ST_PickPlace;
    EmptyTrussInfo : ST_TrussInfo;
    result         : USINT;
END_VAR
IF ConvData[1].State = E_Outfeed_Conveyor_State.IDLE THEN
    FOR i := 1 TO 50 DO
        IF ConvData[1].BoardsPresent[i].ID = '' AND ConvData[1].BoardsPresent[i].Length = 0 THEN
            ConvData[1].BoardsPresent[i] := EmptyBoardData;
        END_IF
    END_FOR

